ABB RAPID module: M_178.mod

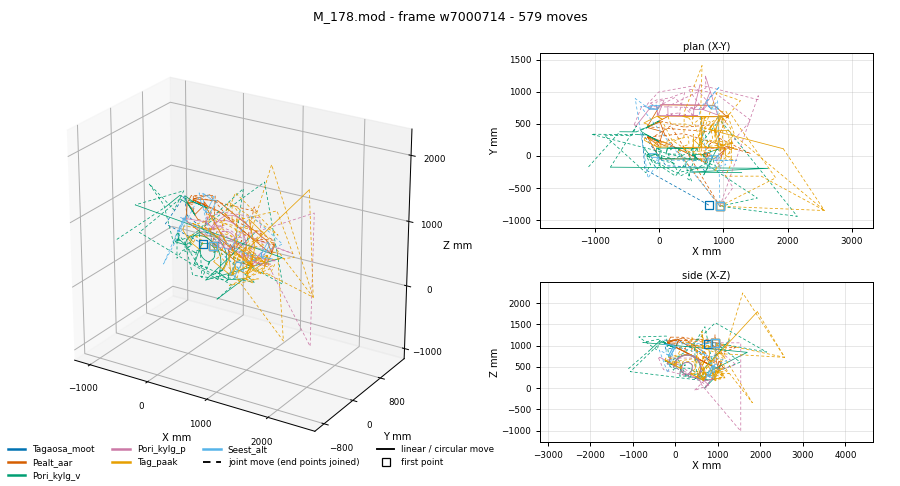
[picture p0: tool path of M_178.mod in frame w7000714, 579 of 583 moves have a stored position in this frame; points joined in program order, loops and branches not executed]
MODULE HITS_P

TASK PERS wobjdata w7000714:=[FALSE,FALSE,"STN2",[[0,0,0],[1,0,0,0]],[[375.036068751363,-383.154606661982,156.369033292662],[0.707106781186547,2.71584596430043E-17,2.9305070426361E-17,0.707106781186548]]];
CONST robtarget mooduli_vahetus := [[944.98,-783.48,1066.49],[0.140873,0.0138616,0.989908,-0.00676465],[0,-1,0,0],[358.608,-0.00699401,0.0391992,9E+09,9E+09,9E+09]];
CONST robtarget mooduli_vahetu10:=[[-90.91,322.81,1276.86],[0.262384,-0.0974996,0.959945,-0.0125037],[0,-1,0,0],[122.138,-6.09681,44.9368,9E+09,9E+09,9E+09]];
CONST robtarget mooduli_vahetu20:=[[3.88,808.65,1089.11],[0.234461,-0.125171,0.933949,-0.238956],[1,-1,0,0],[122.138,-6.09681,44.937,9E+09,9E+09,9E+09]];
TASK PERS pose VE1 := [[-6.83543,-0.0174255,-0.579834],[1,0,0,0]];
TASK PERS pose PE1 := [[0.5466,-0.00140381,0.050415],[1,0,0,0]];
TASK PERS pose VK1 := [[-0.057518,-0.763161,-0.332397],[1,0,0,0]];
TASK PERS pose VK2 := [[0.0793457,0.896591,0.228455],[1,0,0,0]];
TASK PERS pose VKs1 := [[1,2,0],[1,0,0,0]];
TASK PERS pose PEs1 := [[0,3,0],[1,0,0,0]];
TASK PERS pose PE2 := [[0,2,0],[1,0,0,0]];
TASK PERS pose VE2 := [[0,2,0],[1,0,0,0]];
TASK PERS pose VP1 := [[0.214996,0.419937,-0.887817],[1,0,0,0]];

  !**********************************************************
  !
  ! (c) Norcar-BSB Eesti AS
  !
  !**********************************************************
  !
  ! Moodul:       	7000714
  !
  ! Autor:   		Martins, Erki, Kert
  !
  ! Description:  	7000714 a60 tagaosa keevitusprogramm
  !
  ! Protseduurid:   	m??tmine enne keevitust smartac
  !
  ! Funktsioonid:    	m??tmine, keevitamine
  !
  ! Kuup?ev:      	04.03.2010
  !
  ! Versioon:      	0.7
  !
  ! Rakised:		a60 tagaosa rakis
  !
  ! Ajalugu:      	0.1 alustatud proge kirjutamist 04.03.2010
  !                 	0.2 esimene moodul tehtud 29.03.2010
  !				0.3 teine ja kolmas moodul tehtud 31.03.2010
  !				0.4 paagi mooduli tegemine 07.04.2010
  !				0.5 programmi korrastamine 08.04.2010
  !                	0.6 keevitusparameetrid sisse ja katsed 09.04.2010
  !				0.7 teise ringi katsetamine ja viies moodul
  !				0.8
  !
  !************************************************************

PROC HitsPMain()
	ActUnit STN2;
	Reset aDoRobHome;
	DRW_Number:="7000714";
	IF aDiK??ntP?ytOK=0 TPWrite "Waiting for turntables to reach home position";
	WaitDI aDiK??ntP?ytOK,1;

	TPErase;
	TPWrite "Traktori a60 tagaosa keevitus 7000714";
	TPWrite "versioon 0.7, 09.04.2010";

	! Parem pool valida tagant pool vaadates
	! rakise kaldenurk 27,3 kraadi

	! keevitusparameetrid: wld70v12sh24 ?huke plekk
	! weld100v10sh16 porilaud ja ??r kokku, l?hikesed ?mblused
	! wld100v5sh12 kere ja porilaud
	! wld200v10sh14 ots ja kere
	! wld250v6sh11 tugevdusribi
	! weld250v10sh11 korpus ja kaitseraud
	! wld200v6sh16 paksemad plaadid
	! wld200v8sh14 puksid, ring?mblused

start:
TPReadFK reg1,"Tee oma valik","M??da","Keevita","L?peta","","";

IF reg1=1 THEN
       GOTO yks;
ELSEIF reg1=2 THEN
       GOTO alusta;
ELSEIF reg1=3 THEN
       GOTO end;
    ENDIF

yks:
	Tagaosa_moot;
	GOTO start;

alusta:
Stop;

	! Moodul 1
	! Pealt perimeeter ja paagid kokku
	Pealt_aar;

	! Puhastus
	PuhdistRutWeld;

	! Moodul 2
	! Porilaud ja k?ljed vasakult
	!Stop;
	Pori_kylg_v;

	! Puhastus
	PuhdistRutWeld;

	! Moodul 3
	!Stop;
	! Porilaud ja k?ljed paremalt
	Pori_kylg_p;

	! Puhastus
	PuhdistRutWeld;

	! Moodul 4
	! tagaots ja paak seest
	Tag_paak;

	! Puhastus
	PuhdistRutWeld;

	! Moodul 5
	! V?ljast kinnitused ja alt puksid
	!Stop;
	Seest_alt;

	! Puhastus
	PuhdistRutWeld;

	GOTO end;
end:

MoveJ pHomeS2, v500, fine, tPKI500;
    DeactUnit STN2;
    RETURN;
ENDPROC


! M??tmine
PROC Tagaosa_moot()

	Stop;
	MoveJ [[771.19,-764.83,1049.41],[0.17262,-0.011269,0.984924,0.00151479],[0,-1,0,0],[358.606,0.00534949,0.0600025,9E+09,9E+09,9E+09]], v600, z200, tPKI500\WObj:=w7000714;

	! M??tmine smarttaciga ja pdisp kasutamine

	PDispOff;

	! Search - PROOV m??dab tagaosa

	!eest tagasapikkuse m66t
	MoveJ [[-222.07,-210.04,919.03],[0.387473,-0.533268,-0.439373,-0.610281],[1,-1,-2,0],[33.7138,0.00525396,0.0596227,9E+09,9E+09,9E+09]], v600, z200, tPKI500\WObj:=w7000714;
	Search_1D VE1, [[-281.87,349.61,976.70],[0.455775,-0.478529,-0.500064,-0.559657],[0,-1,-2,0],[33.7116,0.00531128,0.0594539,9E+09,9E+09,9E+09]], [[-245.65,349.67,979.75],[0.456433,-0.47783,-0.499358,-0.560349],[0,-1,-2,0],[33.7116,0.00531128,0.0592429,9E+09,9E+09,9E+09]], v600, tPKI500\WObj:=w7000714;
	Search_1D PE1, [[-279.88,515.34,977.24],[0.455844,-0.478471,-0.499981,-0.559725],[0,-1,-2,0],[33.7116,0.00531128,0.0593273,9E+09,9E+09,9E+09]], [[-250.66,515.16,979.95],[0.456426,-0.477841,-0.499362,-0.560342],[0,-1,-2,0],[33.7112,0.00525396,0.0593273,9E+09,9E+09,9E+09]], v600, tPKI500\WObj:=w7000714;
	MoveJ [[-271.44,361.19,1131.71],[0.456425,-0.477848,-0.499367,-0.560332],[0,-1,-2,0],[33.7116,0.00531128,0.0594539,9E+09,9E+09,9E+09]], v600, z200, tPKI500\WObj:=w7000714;

	!Vasaku kulje m66tmine
	MoveJ [[105.72,-153.88,1105.54],[0.108349,-0.674265,0.730311,-0.0165769],[0,0,-1,0],[33.7125,0.00534949,0.0591586,9E+09,9E+09,9E+09]], v600, z200, tPKI500\WObj:=w7000714;
	Search_1D VK1, [[120.39,-78.73,857.25],[0.0242109,0.669444,-0.741611,-0.0356805],[0,0,-1,0],[33.7132,0.00531128,0.0591586,9E+09,9E+09,9E+09]], [[121.03,-69.16,861.51],[0.0222677,0.66942,-0.741686,-0.03584],[0,0,-1,0],[33.7129,0.00534949,0.0591586,9E+09,9E+09,9E+09]], v600, tPKI500\WObj:=w7000714;
	MoveJ [[657.53,-174.78,809.55],[0.0222674,0.669428,-0.741679,-0.0358406],[0,0,-1,0],[33.7119,0.00534949,0.0590742,9E+09,9E+09,9E+09]], v600, z200, tPKI500\WObj:=w7000714;
	Search_1D VK2, [[706.38,-87.21,543.09],[0.0241212,0.669347,-0.74167,-0.0363144],[0,0,-2,0],[33.7125,0.00534949,0.0591586,9E+09,9E+09,9E+09]], [[707.65,-71.68,547.01],[0.0222997,0.669456,-0.741652,-0.0358542],[0,0,-2,0],[33.7125,0.00534949,0.0591586,9E+09,9E+09,9E+09]], v600, tPKI500\WObj:=w7000714;
	MoveJ [[706.29,-234.46,900.27],[0.0223105,0.669463,-0.741645,-0.0358672],[0,0,-1,0],[33.7119,0.00531128,0.0591586,9E+09,9E+09,9E+09]], v600, z200, tPKI500\WObj:=w7000714;
	!
	!
	MoveJ [[706.29,-234.46,900.26],[0.0223165,0.669465,-0.741643,-0.0358642],[0,0,-1,0],[33.7129,0.00531128,0.0592429,9E+09,9E+09,9E+09]], v600, z200, tPKI500\WObj:=w7000714;
	!
	!
	!

ENDPROC


! Pealt perimeeter ja paagid kokku
PROC Pealt_aar()

MoveJ mooduli_vahetus, v600, z50, tPKI500\WObj:=w7000714;

! kallutab lauda 17 kraadi, telg 1
MoveJ [[180.24,469.35,1197.20],[0.0518904,-0.882291,0.437678,0.165258],[0,-2,1,0],[252.909,16.9763,0.0391992,9E+09,9E+09,9E+09]], v200, z50, tPKI500\WObj:=w7000714;

! Keevitus 1.5, pealt sisemine perimeeter, esimene ?mblus, 90 mm, vasakult, OK
MoveJ [[-106.16,285.70,1199.65],[0.365736,0.833576,-0.285271,-0.300015],[0,-2,1,0],[223.84,16.9756,0.0391992,9E+09,9E+09,9E+09]], v600, z50, tPKI500\WObj:=w7000714;
PDispSet VKs1;
ArcLStart [[-184.93,290.61,1062.16],[0.282147,0.91122,-0.00162775,-0.300115],[0,-2,1,0],[223.922,16.9756,0.0353171,9E+09,9E+09,9E+09]], v600, seam1, m178job63, fine, tPKI500\WObj:=w7000714;
ArcL [[-182.70,295.03,1059.96],[0.31567,0.897368,-0.0303764,-0.306858],[0,-1,1,0],[223.905,16.975,0.0354859,9E+09,9E+09,9E+09]], v600, seam1, m178job63, fine, tPKI500\WObj:=w7000714;
ArcL [[-181.16,297.14,1059.57],[0.343632,0.766621,-0.361756,-0.404157],[0,-1,1,0],[223.774,16.9772,0.0418576,9E+09,9E+09,9E+09]], v600, seam1, m178job63, fine, tPKI500\WObj:=w7000714;
ArcLEnd [[-107.54,258.50,1021.43],[0.343541,0.766447,-0.362409,-0.403981],[0,-1,1,0],[223.649,16.975,0.0421108,9E+09,9E+09,9E+09]], v600, seam1, m178job63, fine, tPKI500\WObj:=w7000714;
PDispOff;
!Stop;

! Keevitus 1.6, pealt sisemine perimeeter, teine ?mblus, 170 mm, vasakult, OK
MoveJ [[-21.88,220.27,1045.21],[0.344664,0.764827,-0.363237,-0.405348],[0,-1,1,0],[223.835,16.9754,0.0388194,9E+09,9E+09,9E+09]], v600, z50, tPKI500\WObj:=w7000714;
ArcLStart [[-37.58,223.17,985.34],[0.34387,0.766267,-0.362247,-0.404187],[0,-1,1,0],[223.715,16.9765,0.0378489,9E+09,9E+09,9E+09]], v600, seam1, m178job63, fine, tPKI500\WObj:=w7000714;
ArcLEnd [[83.74,158.59,921.84],[0.344,0.766329,-0.362082,-0.404106],[0,-1,1,0],[223.926,16.9761,0.0403807,9E+09,9E+09,9E+09]], v600, seam1, m178job63, fine, tPKI500\WObj:=w7000714;
MoveJ [[206.18,140.94,924.64],[0.344664,0.764847,-0.363211,-0.405332],[0,-1,1,0],[223.836,16.9754,0.038946,9E+09,9E+09,9E+09]], v600, z50, tPKI500\WObj:=w7000714;

! Keevitus 1.7, pealt sisemine perimeeter, kolmas ?mblus, 900 mm, vasakult, OK
MoveJ [[245.32,122.46,948.22],[0.428788,0.781292,-0.355324,-0.281904],[0,-2,1,0],[223.836,16.9754,0.0390304,9E+09,9E+09,9E+09]], v600, z50, tPKI500\WObj:=w7000714;
ArcLStart [[219.87,127.02,851.73],[0.430441,0.781418,-0.353698,-0.28108],[0,-2,1,0],[223.838,16.9791,0.036583,9E+09,9E+09,9E+09]], v600, seam1, m178job63, fine, tPKI500\WObj:=w7000714;
ArcL [[342.17,127.04,789.47],[0.429347,0.781714,-0.354074,-0.281457],[0,-2,1,0],[223.735,16.9768,0.0410137,9E+09,9E+09,9E+09]], v600, seam1, m178job63, fine, tPKI500\WObj:=w7000714;
ArcL [[409.75,126.28,753.72],[0.429439,0.781537,-0.354188,-0.281664],[0,-2,1,0],[223.879,16.9747,0.039579,9E+09,9E+09,9E+09]], v600, seam1, m178job63, fine, tPKI500\WObj:=w7000714;
ArcL [[602.52,125.87,654.64],[0.429815,0.781282,-0.354003,-0.28203],[0,-2,1,0],[223.76,16.9766,0.0403807,9E+09,9E+09,9E+09]], v600, seam1, m178job63, fine, tPKI500\WObj:=w7000714;
ArcL [[895.88,124.47,502.15],[0.430572,0.780641,-0.353814,-0.282886],[0,-2,1,0],[223.711,16.9752,0.0383975,9E+09,9E+09,9E+09]], v600, seam1, m178job63, fine, tPKI500\WObj:=w7000714;
ArcLEnd [[1023.79,124.57,438.15],[0.316212,0.827255,-0.461489,-0.0518623],[0,-2,1,0],[223.957,16.9767,0.0422796,9E+09,9E+09,9E+09]], v600, seam1, m178job63, fine, tPKI500\WObj:=w7000714;
!Stop;
MoveL [[964.69,-11.95,633.96],[0.365253,0.816264,-0.423133,-0.145816],[0,-2,1,0],[223.84,16.9754,0.0391148,9E+09,9E+09,9E+09]], v600, z50, tPKI500\WObj:=w7000714;
MoveJ [[935.24,302.49,1253.35],[0.268514,0.719805,-0.421181,-0.482067],[0,-2,1,0],[900.475,16.9763,0.038946,9E+09,9E+09,9E+09]], v600, z50, tPKI500\WObj:=w7000714;

! tagaosa liigutamine, p??ramine -180 ja kallutamine -17 kraadi
MoveJ [[933.23,364.67,1157.80],[0.156036,0.433261,-0.854217,-0.241355],[0,0,0,0],[900.473,0.0294633,-0.0224089,9E+09,9E+09,9E+09]], v200, z50, tPKI500\WObj:=w7000714;


! Keevitus 1.8, pealt sisemine perimeeter, 400+1000 mm, paremalt, OK
MoveJ [[-182.46,453.50,1113.53],[0.0239912,-0.818382,-0.566844,-0.0914538],[0,0,-1,0],[900.473,-17.0628,-180.01,9E+09,9E+09,9E+09]], v600, z50, tPKI500\WObj:=w7000714;
!PDispSet PEs1;
ArcLStart [[-181.60,450.94,1062.98],[0.503117,-0.413223,-0.733358,0.195723],[0,0,-2,0],[900.45,-17.0603,-180.002,9E+09,9E+09,9E+09]], v600, seam1, m178job63, fine, tPKI500\WObj:=w7000714;
ArcL [[145.59,620.57,892.53],[0.508981,-0.543619,-0.650043,0.151203],[0,-1,-1,0],[900.468,-17.0623,-180.011,9E+09,9E+09,9E+09]], v600, seam1, m178job63, fine, tPKI500\WObj:=w7000714;
!PDispOff;
ArcL [[189.40,619.81,872.09],[0.508359,-0.544165,-0.649758,0.152549],[0,-1,-1,0],[900.389,-17.0611,-180.01,9E+09,9E+09,9E+09]], v600, seam1, m178job63, fine, tPKI500\WObj:=w7000714;
ArcL [[963.08,613.27,470.38],[0.507653,-0.544392,-0.649926,0.153374],[1,-1,0,0],[900.441,-17.0625,-180.009,9E+09,9E+09,9E+09]], v600, seam1, m178job63, fine, tPKI500\WObj:=w7000714;
ArcLEnd [[1025.00,613.30,438.63],[0.324043,-0.564722,-0.758986,0.00524122],[1,-1,0,0],[900.51,-17.0616,-180.01,9E+09,9E+09,9E+09]], v600, seam1, m178job63, fine, tPKI500\WObj:=w7000714;
MoveL [[1079.67,612.90,617.47],[0.409142,-0.560838,-0.716391,0.0696263],[1,-1,0,0],[900.466,-17.0627,-180.01,9E+09,9E+09,9E+09]], v600, z50, tPKI500\WObj:=w7000714;
MoveJ [[819.08,483.11,649.57],[0.380352,-0.742193,-0.550233,-0.0415458],[1,-1,0,0],[900.473,-17.0628,-180.01,9E+09,9E+09,9E+09]], v600, z50, tPKI500\WObj:=w7000714;
!Stop;

! Keevitus 1.9, pealt v?limine perimeeter, 400+960+260 mm, paremalt, OK
MoveJ [[384.40,449.47,940.53],[0.521441,-0.593526,-0.607333,0.0835091],[1,-1,-1,0],[900.473,-17.0628,-180.01,9E+09,9E+09,9E+09]], v600, z50, tPKI500\WObj:=w7000714;
MoveJ [[46.17,534.77,1158.25],[0.600818,-0.379123,-0.690069,0.138168],[0,0,-2,0],[900.473,-25.7634,-166.314,9E+09,9E+09,9E+09]], v600, z50, tPKI500\WObj:=w7000714;
!PDispSet PE2;
!Stop;
ArcLStart [[-184.51,460.44,1069.91],[0.496644,-0.128395,-0.848,0.133251],[0,0,-2,0],[900.771,-25.7553,-166.306,9E+09,9E+09,9E+09]], v600, seam1, m178job64, fine, tPKI500\WObj:=w7000714;
ArcL [[-173.78,476.50,1064.44],[0.554302,-0.193481,-0.808682,0.0367356],[0,0,-2,0],[900.416,-25.7545,-166.312,9E+09,9E+09,9E+09]], v600, seam1, m178job64, fine, tPKI500\WObj:=w7000714;
ArcL [[7.04,779.24,972.40],[0.572647,-0.266003,-0.772129,0.071665],[0,0,-2,0],[900.468,-25.7619,-166.314,9E+09,9E+09,9E+09]], v600, seam1, m178job64, fine, tPKI500\WObj:=w7000714;
ArcL [[16.15,792.14,969.22],[0.546633,-0.32251,-0.771885,-0.0370876],[0,0,-2,0],[900.605,-25.7608,-166.312,9E+09,9E+09,9E+09]], v600, seam1, m178job64, fine, tPKI500\WObj:=w7000714;
ArcL [[17.29,792.63,968.97],[0.486097,-0.575984,-0.655473,-0.0480558],[0,0,-1,0],[900.465,-25.7615,-166.313,9E+09,9E+09,9E+09]], v600, seam1, m178job64, fine, tPKI500\WObj:=w7000714;
ArcL [[61.54,794.51,942.69],[0.486117,-0.575989,-0.655457,-0.0479974],[0,0,-1,0],[900.479,-25.7614,-166.313,9E+09,9E+09,9E+09]], v600, seam1, m178job64, fine, tPKI500\WObj:=w7000714;
!ArcL [[26.13,798.11,960.35],[0.484105,-0.561883,-0.669531,0.0407281],[0,0,-2,0],[900.564,-25.7615,-166.313,9E+09,9E+09,9E+09]], v600, seam1, m178job64, fine, tPKI500\WObj:=w7000714;
!PDispOff;
ArcL [[218.26,793.40,860.22],[0.440223,-0.59926,-0.666261,-0.0564766],[0,0,-1,0],[900.512,-22.7548,-167.365,9E+09,9E+09,9E+09]], v600, seam1, m178job64, fine, tPKI500\WObj:=w7000714;
ArcL [[462.67,790.42,734.13],[0.443653,-0.60729,-0.65239,-0.0935942],[0,0,-1,0],[900.43,-22.7561,-167.369,9E+09,9E+09,9E+09]], v600, seam1, m178job64, fine, tPKI500\WObj:=w7000714;
ArcL [[742.57,789.03,587.93],[0.462626,-0.587719,-0.662256,-0.0445244],[1,-1,-1,0],[900.527,-22.7574,-167.369,9E+09,9E+09,9E+09]], v600, seam1, m178job64, fine, tPKI500\WObj:=w7000714;
ArcL [[851.66,788.32,531.91],[0.452915,-0.692054,-0.556899,-0.0761225],[1,-1,0,0],[900.414,-22.756,-167.367,9E+09,9E+09,9E+09]], v600, seam1, m178job64, fine, tPKI500\WObj:=w7000714;
ArcL [[855.89,786.75,530.12],[0.309039,-0.756387,-0.542731,-0.194471],[1,-1,0,0],[900.592,-22.7566,-167.369,9E+09,9E+09,9E+09]], v600, seam1, m178job64, fine, tPKI500\WObj:=w7000714;
ArcL [[865.09,778.53,525.36],[0.240514,-0.776627,-0.559111,-0.162482],[1,-1,0,0],[900.34,-22.7565,-167.369,9E+09,9E+09,9E+09]], v600, seam1, m178job64, fine, tPKI500\WObj:=w7000714;
ArcL [[1023.44,637.84,443.03],[0.305172,-0.843887,-0.420352,-0.13428],[1,-1,0,0],[900.508,-21.6371,-168.17,9E+09,9E+09,9E+09]], v600, seam1, m178job64, fine, tPKI500\WObj:=w7000714;
ArcLEnd [[1028.26,628.31,439.23],[0.104333,-0.92647,-0.329608,-0.148755],[1,-1,1,0],[900.435,-21.637,-168.167,9E+09,9E+09,9E+09]], v600, seam1, m178job64, fine, tPKI500\WObj:=w7000714;
MoveL [[1077.12,631.65,580.85],[0.334968,-0.898779,-0.276011,-0.0617454],[1,-1,0,0],[900.462,-17.0628,-180.01,9E+09,9E+09,9E+09]], v600, z50, tPKI500\WObj:=w7000714;
!Stop;
MoveJ [[911.67,287.97,765.35],[0.263835,-0.727529,-0.625551,0.0988923],[1,-1,0,0],[900.476,-17.0627,-180.01,9E+09,9E+09,9E+09]], v600, z50, tPKI500\WObj:=w7000714;

!laua pooramine 0?;0? ja puhastus
MoveJ [[1416.30,39.74,954.05],[0.0989373,0.157025,-0.973447,0.134],[0,-1,0,0],[900.477,0.118753,0.0317303,9E+09,9E+09,9E+09]], v200, z50, tPKI500\WObj:=w7000714;
PuhdistRutWeld;

! laua p??ramine 0 ja 17 kraadi
MoveJ [[373.90,347.34,998.41],[0.117153,0.675178,-0.725187,0.0672047],[1,-1,0,0],[900.477,17.0189,0.0317303,9E+09,9E+09,9E+09]], v200, z50, tPKI500\WObj:=w7000714;

! Keevitus 1.16, pealt v?limine perimeeter, katkestusega, 400+960+260 mm, vasakult, OK
MoveJ [[-90.42,300.54,1139.12],[0.392371,0.593922,-0.666197,-0.222452],[1,-1,0,0],[900.477,17.0189,0.0318147,9E+09,9E+09,9E+09]], v600, z50, tPKI500\WObj:=w7000714;
MoveJ [[-7.26,155.27,1132.10],[0.55973,0.636495,-0.490279,-0.202987],[1,-1,1,0],[900.477,23.261,-19.6927,9E+09,9E+09,9E+09]], v600, z50, tPKI500\WObj:=w7000714;
!PDispSet VE2;
ArcLStart [[-180.99,293.89,1069.89],[0.361586,0.702678,-0.482614,-0.377604],[1,-2,1,0],[900.55,23.2609,-19.6886,9E+09,9E+09,9E+09]], v600, seam1, m178job64, fine, tPKI500\WObj:=w7000714;
ArcL [[-172.19,275.51,1065.82],[0.362528,0.703271,-0.480746,-0.377979],[1,-2,1,0],[900.472,23.2629,-19.6841,9E+09,9E+09,9E+09]], v600, seam1, m178job64, fine, tPKI500\WObj:=w7000714;
ArcL [[12.62,-41.24,969.35],[0.363305,0.702574,-0.478589,-0.381252],[1,-2,1,0],[900.464,23.2617,-19.681,9E+09,9E+09,9E+09]], v600, seam1, m178job64, fine, tPKI500\WObj:=w7000714;
ArcL [[13.93,-43.98,966.67],[0.490227,0.715866,-0.473325,-0.152242],[1,-1,1,0],[900.529,23.2631,-19.6823,9E+09,9E+09,9E+09]], v600, seam1, m178job64, fine, tPKI500\WObj:=w7000714;
ArcL [[17.76,-45.14,963.78],[0.490161,0.716042,-0.473108,-0.152305],[1,-1,1,0],[900.405,23.263,-19.6888,9E+09,9E+09,9E+09]], v600, seam1, m178job64, fine, tPKI500\WObj:=w7000714;
!PDispOff;
ArcL [[409.73,-46.28,760.58],[0.489184,0.715938,-0.472985,-0.15626],[1,-1,0,0],[900.468,23.2622,-19.688,9E+09,9E+09,9E+09]], v600, seam1, m178job64, fine, tPKI500\WObj:=w7000714;
ArcL [[452.01,-46.08,738.89],[0.489114,0.71587,-0.473171,-0.156229],[1,-1,0,0],[900.642,23.2626,-19.6822,9E+09,9E+09,9E+09]], v600, seam1, m178job64, fine, tPKI500\WObj:=w7000714;
ArcL [[837.00,-47.76,538.25],[0.479378,0.722246,-0.473393,-0.156391],[0,0,-1,0],[900.538,23.2626,-19.6881,9E+09,9E+09,9E+09]], v600, seam1, m178job64, fine, tPKI500\WObj:=w7000714;
ArcL [[851.61,-46.66,530.84],[0.423876,0.859284,-0.254656,-0.13081],[0,0,-1,0],[900.402,23.2616,-19.691,9E+09,9E+09,9E+09]], v600, seam1, m178job64, fine, tPKI500\WObj:=w7000714;
ArcL [[857.00,-42.95,528.28],[0.386827,0.86793,-0.301478,-0.0785747],[0,0,-1,0],[900.62,20.2871,-19.3544,9E+09,9E+09,9E+09]], v600, seam1, m178job64, fine, tPKI500\WObj:=w7000714;
ArcL [[1012.18,92.00,448.44],[0.339783,0.9362,-0.0832581,-0.0338601],[0,0,-1,0],[900.49,20.2809,-19.3547,9E+09,9E+09,9E+09]], v600, seam1, m178job64, fine, tPKI500\WObj:=w7000714;
ArcL [[1023.90,103.83,443.36],[0.30711,0.951266,0.025384,-0.0115288],[0,0,-1,0],[900.508,20.2817,-19.3543,9E+09,9E+09,9E+09]], v600, seam1, m178job64, fine, tPKI500\WObj:=w7000714;
ArcLEnd [[1028.97,114.26,441.04],[0.30716,0.951259,0.0250954,-0.011467],[0,0,-1,0],[900.484,20.2805,-19.3551,9E+09,9E+09,9E+09]], v600, seam1, m178job64, fine, tPKI500\WObj:=w7000714;
MoveJ [[1009.60,129.26,607.74],[0.344702,0.916928,-0.125824,-0.156824],[0,0,-1,0],[900.477,17.0188,0.0318147,9E+09,9E+09,9E+09]], v600, z50, tPKI500\WObj:=w7000714;
GOTO toruta;

! laua kallutamine 27,3 kraadi
MoveJ [[1162.57,122.71,472.36],[0.140864,0.966293,-0.206823,0.0605097],[0,0,-1,0],[900.479,27.2716,0.0316459,9E+09,9E+09,9E+09]], v200, z50, tPKI500\WObj:=w7000714;

! Keevitus 1.17, paagi ?litoru keevitus, D65, 205 mm, vasakult, OK
MoveJ [[761.07,123.30,678.14],[0.365414,0.711061,-0.597258,0.0644121],[1,-1,0,0],[900.479,27.2716,0.0317303,9E+09,9E+09,9E+09]], v600, z50, tPKI500\WObj:=w7000714;
MoveJ [[796.44,199.49,743.61],[0.0479302,0.973161,-0.128236,0.184981],[0,0,-2,0],[380.209,27.2717,0.0316459,9E+09,9E+09,9E+09]], v600, z50, tPKI500\WObj:=w7000714;
MoveJ [[687.10,23.33,635.41],[0.047942,0.973163,-0.128221,0.184975],[0,0,-2,0],[380.21,27.2717,0.0317303,9E+09,9E+09,9E+09]], v600, z50, tPKI500\WObj:=w7000714;
ArcLStart [[695.23,20.35,610.24],[0.0479757,0.973171,-0.128186,0.184952],[0,0,-2,0],[380.209,27.2718,0.0316459,9E+09,9E+09,9E+09]], v600, seam1, wld200v8sh14, fine, tPKI500\WObj:=w7000714;
ArcC [[703.68,41.46,605.91],[0.233173,0.884181,-0.372829,0.157648],[0,0,-1,0],[380.209,27.2718,0.0315615,9E+09,9E+09,9E+09]], [[724.22,51.48,595.17],[0.413668,0.677563,-0.590079,0.146955],[0,0,-1,0],[380.209,27.2717,0.0317303,9E+09,9E+09,9E+09]], v600, seam1, wld200v8sh14, fine, tPKI500\WObj:=w7000714;
ArcC [[744.31,37.77,584.31],[0.560827,0.279575,-0.774777,0.0838623],[0,-1,0,0],[380.211,27.2717,0.0318991,9E+09,9E+09,9E+09]], [[749.01,21.17,581.66],[0.605493,-0.100927,-0.789225,0.0178112],[0,-1,0,0],[380.211,27.2717,0.0319835,9E+09,9E+09,9E+09]], v600, seam1, wld200v8sh14, fine, tPKI500\WObj:=w7000714;
ArcC [[738.53,-3.73,586.77],[0.523729,-0.550732,-0.646299,-0.068564],[0,-1,1,0],[380.211,27.2717,0.0317303,9E+09,9E+09,9E+09]], [[720.80,-10.17,596.10],[0.382247,-0.798907,-0.44818,-0.121536],[0,-1,1,0],[380.209,27.2717,0.0318147,9E+09,9E+09,9E+09]], v600, seam1, wld200v8sh14, fine, tPKI500\WObj:=w7000714;
ArcCEnd [[702.53,-1.70,606.23],[0.217979,-0.937243,-0.220726,-0.159192],[0,0,2,0],[380.209,27.2717,0.0317303,9E+09,9E+09,9E+09]], [[694.97,21.51,610.10],[0.0305759,-0.983588,0.026777,-0.175798],[0,0,2,0],[380.209,27.2717,0.0318991,9E+09,9E+09,9E+09]], v600, seam1, wld200v8sh14, fine, tPKI500\WObj:=w7000714;
MoveJ [[677.39,22.28,657.51],[0.0305932,-0.983584,0.0267976,-0.175812],[0,0,2,0],[380.21,27.2717,0.0317303,9E+09,9E+09,9E+09]], v600, z50, tPKI500\WObj:=w7000714;
MoveJ [[715.23,21.87,731.36],[0.0314181,-0.983594,0.0257474,-0.175765],[0,0,2,0],[380.212,27.2718,0.0315615,9E+09,9E+09,9E+09]], v600, z50, tPKI500\WObj:=w7000714;

! keevitus 1.18 olitoru 2. keevitus. Sihtida korgemale.
ArcLStart [[748.47,20.52,697.24],[0.0284428,-0.989467,0.0292656,-0.138894],[0,0,2,0],[380.211,27.2719,0.0312661,9E+09,9E+09,9E+09]], v600, seam1, wld100v5sh12, fine, tPKI500\WObj:=w7000714;
ArcC [[753.90,3.52,693.53],[0.29512,-0.905936,-0.262022,-0.153394],[0,0,2,0],[380.212,27.2719,0.0314771,9E+09,9E+09,9E+09]], [[758.04,0.42,692.07],[0.378817,-0.848515,-0.341376,-0.141365],[0,0,1,0],[380.213,27.2719,0.0315615,9E+09,9E+09,9E+09]], v600, seam1, wld100v5sh12, fine, tPKI500\WObj:=w7000714;
ArcC [[780.52,-0.11,681.16],[0.555558,-0.48452,-0.674518,-0.0402726],[0,-1,1,0],[380.212,27.272,0.0314771,9E+09,9E+09,9E+09]], [[789.68,16.12,677.29],[0.605207,-0.15056,-0.780951,0.034251],[0,-1,0,0],[380.212,27.2721,0.0315615,9E+09,9E+09,9E+09]], v600, seam1, wld100v5sh12, fine, tPKI500\WObj:=w7000714;
ArcC [[782.12,40.39,684.13],[0.48532,0.491825,-0.717743,0.086131],[0,-1,0,0],[380.215,27.2721,0.0316459,9E+09,9E+09,9E+09]], [[766.85,42.10,690.36],[0.2943,0.775359,-0.532609,0.168922],[0,0,-1,0],[380.214,27.272,0.0316459,9E+09,9E+09,9E+09]], v600, seam1, wld100v5sh12, fine, tPKI500\WObj:=w7000714;
ArcCEnd [[752.38,30.72,696.63],[0.0823334,0.954908,-0.245845,0.144683],[0,0,-2,0],[380.213,27.272,0.0317303,9E+09,9E+09,9E+09]], [[749.81,18.20,698.25],[0.0187265,-0.982495,0.0795466,-0.167411],[0,0,-2,0],[380.209,27.2719,0.0316459,9E+09,9E+09,9E+09]], v600, seam1, wld100v5sh12, fine, tPKI500\WObj:=w7000714;
MoveJ [[725.98,-104.59,807.21],[0.0243497,-0.967141,0.0782152,-0.240685],[0,0,-2,0],[380.212,27.2719,0.0312661,9E+09,9E+09,9E+09]], v600, z50, tPKI500\WObj:=w7000714;

! manualis aeg 13:55, 100% kiirusel
toruta:
MoveL [[188.78,164.77,1182.32],[0.351757,0.903929,-0.102661,-0.220549],[1,0,-1,0],[900.477,24.9716,0.185371,9E+09,9E+09,9E+09]], v600, z50, tPKI500\WObj:=w7000714;
MoveL [[-169.35,308.67,1074.09],[0.0381361,0.973148,-0.0686915,-0.21636],[1,0,-1,0],[601.879,24.9739,0.1844,9E+09,9E+09,9E+09]], v600, z50, tPKI500\WObj:=w7000714;
!ArcLStart [[-183.69,306.62,1059.10],[0.216625,0.952263,-0.0566688,-0.207508],[1,0,-1,0],[601.881,24.9747,0.183134,9E+09,9E+09,9E+09]], v600, seam1, m178job65, fine, tPKI500\WObj:=w7000714;
!ArcLEnd [[2.47,207.72,962.29],[0.21669,0.952252,-0.0566252,-0.2075],[1,0,-1,0],[601.881,24.9755,0.18229,9E+09,9E+09,9E+09]], v600, seam1, m178job65, fine, tPKI500\WObj:=w7000714;
ArcLStart [[-182.87,310.51,1063.00],[0.119162,0.96529,-0.078063,-0.218912],[1,0,-1,0],[601.92,24.9753,0.18305,9E+09,9E+09,9E+09]], v600, seam1, m178job66, fine, tPKI500\WObj:=w7000714;
ArcLEnd [[6.15,210.21,963.61],[0.119106,0.965289,-0.0780147,-0.218965],[1,0,-1,0],[601.876,24.9747,0.183134,9E+09,9E+09,9E+09]], v600, seam1, m178job66, fine, tPKI500\WObj:=w7000714;
MoveL [[57.63,376.88,1060.42],[0.0744618,-0.973587,0.0548019,0.208764],[1,0,-2,0],[601.885,24.9742,0.184189,9E+09,9E+09,9E+09]], v600, z50, tPKI500\WObj:=w7000714;
!ArcLStart [[-183.72,439.06,1060.86],[0.0763297,-0.957028,0.0605975,0.273131],[1,0,-2,0],[601.907,24.976,0.184189,9E+09,9E+09,9E+09]], v600, seam1, m178job65, fine, tPKI500\WObj:=w7000714;
!ArcLEnd [[8.45,537.87,962.35],[0.07636,-0.957023,0.0606505,0.273127],[1,0,-2,0],[601.862,24.9747,0.185075,9E+09,9E+09,9E+09]], v600, seam1, m178job65, fine, tPKI500\WObj:=w7000714;
ArcLStart [[-182.22,441.27,1061.82],[0.0764125,-0.957017,0.0606314,0.273139],[1,0,-2,0],[601.961,24.9744,0.184527,9E+09,9E+09,9E+09]], v600, seam1, m178job66, fine, tPKI500\WObj:=w7000714;
ArcLEnd [[8.78,538.10,964.11],[0.076471,-0.957017,0.0606792,0.27311],[1,0,-2,0],[601.869,24.9748,0.183683,9E+09,9E+09,9E+09]], v600, seam1, m178job66, fine, tPKI500\WObj:=w7000714;
MoveL [[83.51,335.92,1126.36],[0.0768622,-0.956981,0.0607954,0.273103],[1,0,-2,0],[601.886,24.9746,0.183683,9E+09,9E+09,9E+09]], v600, z50, tPKI500\WObj:=w7000714;

MoveJ mooduli_vahetus, v600, z50, tPKI500\WObj:=w7000714;

ENDPROC


! Porilaud ja k?ljed vasakult
PROC Pori_kylg_v()

MoveJ mooduli_vahetus, v600, z50, tPKI500\WObj:=w7000714;

! laua p??ramine ja kallutamine, -90 ja -90 kraadi
MoveJ [[1527.56,-656.12,612.18],[0.566224,-0.414194,0.434686,0.564697],[0,-1,0,0],[358.609,-90.0158,-89.9705,9E+09,9E+09,9E+09]], v200, z50, tPKI500\WObj:=w7000714;

!alternatiivne porilaua keevitus.2.1
!Stop;
MoveJ [[572.96,-23.79,219.28],[0.459065,0.157412,-0.452009,-0.748445],[0,0,1,0],[358.617,-127.415,-89.6268,9E+09,9E+09,9E+09]], v200, z50, tPKI500\WObj:=w7000714;
ArcLStart [[534.08,14.60,253.95],[0.341392,0.170853,-0.504174,-0.774642],[0,0,1,0],[358.631,-127.415,-89.6265,9E+09,9E+09,9E+09]], v200, seam1, m178job67, fine, tPKI500\WObj:=w7000714;
ArcL [[556.25,-7.26,298.85],[0.341411,0.170778,-0.504216,-0.774623],[0,0,1,0],[358.607,-127.415,-89.6273,9E+09,9E+09,9E+09]], v200, seam1, m178job67, z50, tPKI500\WObj:=w7000714;
ArcL [[570.60,-22.33,326.15],[0.398708,0.10403,-0.486785,-0.770228],[0,0,1,0],[358.715,-125.025,-89.9773,9E+09,9E+09,9E+09]], v200, seam1, m178job67, z50, tPKI500\WObj:=w7000714;
ArcL [[590.63,-49.24,379.80],[0.300559,0.14792,-0.535628,-0.77517],[0,-1,1,0],[358.605,-125.008,-89.9726,9E+09,9E+09,9E+09]], v200, seam1, m178job67, z50, tPKI500\WObj:=w7000714;
ArcC [[597.94,-49.71,418.79],[0.286569,0.224149,-0.674233,-0.642687],[0,-1,1,0],[358.865,-104.881,-89.9757,9E+09,9E+09,9E+09]], [[598.61,-48.93,423.22],[0.284227,0.232138,-0.688042,-0.62604],[0,-1,1,0],[358.894,-102.63,-89.9763,9E+09,9E+09,9E+09]], v200, seam1, m178job67, z10, tPKI500\WObj:=w7000714;
ArcL [[602.32,-49.42,456.59],[0.314306,0.226082,-0.727143,-0.566889],[0,-1,1,0],[358.818,-90.0107,-89.974,9E+09,9E+09,9E+09]], v200, seam1, m178job67, z50, tPKI500\WObj:=w7000714;
ArcC [[583.65,-49.46,578.79],[0.160275,0.384548,-0.734707,-0.535389],[0,-1,1,0],[358.582,-90.0143,-89.9725,9E+09,9E+09,9E+09]], [[558.64,-47.82,631.38],[0.0916303,0.457456,-0.72589,-0.505395],[0,-1,1,0],[358.474,-90.0159,-89.9718,9E+09,9E+09,9E+09]], v200, seam1, m178job67, z10, tPKI500\WObj:=w7000714;
ArcC [[500.41,-48.22,704.55],[0.0154446,0.508368,-0.70911,-0.488352],[0,-1,1,0],[414.039,-90.0124,-89.9729,9E+09,9E+09,9E+09]], [[472.91,-49.06,728.10],[0.0130383,-0.528015,0.7,0.480657],[0,-1,1,0],[435.496,-90.0111,-89.9733,9E+09,9E+09,9E+09]], v200, seam1, m178job67, z10, tPKI500\WObj:=w7000714;
ArcL [[432.66,-46.01,752.17],[0.0667774,-0.558399,0.73443,0.379927],[0,-1,0,0],[443.011,-90.005,-89.9756,9E+09,9E+09,9E+09]], v200, seam1, m178job67, z50, tPKI500\WObj:=w7000714;
ArcC [[320.15,-46.42,786.93],[0.271762,-0.637158,0.678161,0.245507],[0,-1,0,0],[598.731,-90.0089,-89.9756,9E+09,9E+09,9E+09]], [[256.16,-45.59,788.22],[0.37078,-0.666657,0.626103,0.161513],[0,-1,0,0],[683.013,-90.011,-89.9755,9E+09,9E+09,9E+09]], v200, seam1, m178job67, z10, tPKI500\WObj:=w7000714;
ArcC [[183.61,-45.05,773.57],[0.459894,-0.686265,0.559954,0.0631717],[0,-1,0,0],[737.214,-90.0087,-89.9733,9E+09,9E+09,9E+09]], [[151.34,-43.43,760.98],[0.496966,-0.690827,0.524923,0.0154951],[0,-1,0,0],[762.548,-90.0076,-89.9722,9E+09,9E+09,9E+09]], v200, seam1, m178job67, z10, tPKI500\WObj:=w7000714;
ArcL [[104.73,-43.35,735.62],[0.496966,-0.690809,0.524948,0.0154404],[0,-1,0,0],[762.508,-90.0073,-89.9752,9E+09,9E+09,9E+09]], v200, seam1, m178job67, z50, tPKI500\WObj:=w7000714;
ArcC [[66.14,-43.24,707.43],[0.496896,-0.690774,0.525064,0.0153374],[0,-1,0,0],[762.523,-90.0076,-89.9751,9E+09,9E+09,9E+09]], [[29.74,-43.29,672.73],[0.496859,-0.690741,0.525143,0.0152965],[0,-1,0,0],[762.539,-90.0081,-89.975,9E+09,9E+09,9E+09]], v200, seam1, m178job67, z10, tPKI500\WObj:=w7000714;
ArcL [[26.42,-42.31,669.24],[0.575143,-0.706885,0.402383,-0.0872576],[0,-1,0,0],[762.391,-90.0085,-89.9797,9E+09,9E+09,9E+09]], v200, seam1, m178job67, z50, tPKI500\WObj:=w7000714;
ArcL [[-15.58,-9.41,605.64],[0.651434,-0.649324,0.372356,-0.123953],[0,-1,0,0],[762.375,-90.004,-89.9733,9E+09,9E+09,9E+09]], v200, seam1, m178job67, z50, tPKI500\WObj:=w7000714;
ArcLEnd [[-44.01,20.11,549.48],[0.627735,-0.674263,0.358668,-0.150587],[0,-1,0,0],[762.392,-90.0026,-89.9697,9E+09,9E+09,9E+09]], v200, seam1, m178job67, fine, tPKI500\WObj:=w7000714;
MoveJ [[-43.22,8.74,449.30],[0.663991,-0.6342,0.351128,-0.183348],[0,-1,0,0],[776.94,-90.0134,-89.9686,9E+09,9E+09,9E+09]], v200, z50, tPKI500\WObj:=w7000714;

MoveJ [[242.40,-118.53,544.35],[0.758664,-0.445906,0.0707378,-0.469674],[1,0,-1,0],[1427.62,-100.045,-85.4322,9E+09,9E+09,9E+09]], v600, fine, tPKI500\WObj:=w7000714;

! Keevitus 2.3, porilaud seest, 1210 mm, vasakult, OK
MoveJ [[37.81,-70.37,544.52],[0.716966,-0.0163454,-0.364518,-0.593987],[0,0,-2,0],[1009,-90.0122,-89.97,9E+09,9E+09,9E+09]], v600, fine, tPKI500\WObj:=w7000714;
MoveJ [[29.04,84.36,539.17],[0.507124,0.0969799,-0.48977,-0.70253],[0,0,-2,0],[1085.24,-90.0121,-89.97,9E+09,9E+09,9E+09]], v600, fine, tPKI500\WObj:=w7000714;
!Stop;
ArcLStart [[-29.88,122.94,542.89],[0.504484,0.0907541,-0.494967,-0.701618],[0,0,-2,0],[1085.24,-90.0122,-89.9713,9E+09,9E+09,9E+09]], v600, seam1, m178job68, fine, tPKI500\WObj:=w7000714;
ArcL [[10.00,122.87,621.62],[0.483251,0.0799276,-0.492671,-0.719275],[0,0,-2,0],[1085.24,-90.0122,-89.971,9E+09,9E+09,9E+09]], v600, seam1, m178job68, fine, tPKI500\WObj:=w7000714;
ArcC [[58.75,122.93,685.64],[0.485228,0.0583463,-0.513626,-0.705223],[0,0,-2,0],[1046.34,-90.0099,-89.9742,9E+09,9E+09,9E+09]], [[119.77,122.89,733.03],[0.491958,0.0421263,-0.533135,-0.687002],[0,0,-2,0],[1009,-90.0077,-89.9771,9E+09,9E+09,9E+09]], v600, seam1, m178job68, fine, tPKI500\WObj:=w7000714;
ArcC [[180.45,123.46,760.70],[0.564952,-0.058518,-0.45451,-0.686169],[0,0,-2,0],[1009,-90.0078,-89.9767,9E+09,9E+09,9E+09]], [[248.98,123.84,773.44],[0.628969,-0.163144,-0.360116,-0.669403],[0,0,-2,0],[1009,-90.0079,-89.9763,9E+09,9E+09,9E+09]], v600, seam1, m178job68, fine, tPKI500\WObj:=w7000714;
ArcC [[288.93,122.02,772.85],[0.647366,-0.19692,-0.324973,-0.660706],[0,0,-2,0],[1009,-90.0078,-89.9753,9E+09,9E+09,9E+09]], [[407.44,119.21,745.66],[0.691447,-0.299742,-0.217746,-0.620197],[0,0,-2,0],[1009,-90.0075,-89.9721,9E+09,9E+09,9E+09]], v600, seam1, m178job68, fine, tPKI500\WObj:=w7000714;
ArcL [[430.64,118.55,732.15],[0.691541,-0.296732,-0.21608,-0.622119],[0,0,-2,0],[1009,-90.0089,-89.9643,9E+09,9E+09,9E+09]], v600, seam1, m178job68, fine, tPKI500\WObj:=w7000714;
ArcL [[449.20,117.99,721.39],[0.699511,-0.322333,-0.187062,-0.60975],[0,0,-2,0],[1009,-90.0066,-89.9709,9E+09,9E+09,9E+09]], v600, seam1, m178job68, fine, tPKI500\WObj:=w7000714;
ArcC [[523.13,117.92,653.04],[0.717041,-0.389593,-0.103125,-0.568715],[0,0,-2,0],[1008.99,-90.0068,-89.9729,9E+09,9E+09,9E+09]], [[564.33,117.24,586.33],[0.724479,-0.438735,-0.0377625,-0.530299],[0,0,-1,0],[1008.99,-90.0068,-89.9745,9E+09,9E+09,9E+09]], v600, seam1, m178job68, fine, tPKI500\WObj:=w7000714;
ArcC [[582.55,117.02,535.79],[0.717174,-0.48665,0.0381723,-0.49737],[0,0,-1,0],[1008.99,-90.0077,-89.9739,9E+09,9E+09,9E+09]], [[591.35,116.37,447.22],[0.688918,-0.560779,0.158604,-0.431005],[0,0,-1,0],[1009,-90.0093,-89.9725,9E+09,9E+09,9E+09]], v600, seam1, m178job68, fine, tPKI500\WObj:=w7000714;
ArcC [[590.62,117.25,433.10],[0.684383,-0.575368,0.18668,-0.407092],[0,0,-1,0],[1009,-90.0097,-89.9724,9E+09,9E+09,9E+09]], [[578.25,117.74,373.69],[0.651778,-0.626599,0.305234,-0.298987],[0,-1,-1,0],[1009,-90.0111,-89.9718,9E+09,9E+09,9E+09]], v600, seam1, m178job68, fine, tPKI500\WObj:=w7000714;
ArcL [[565.13,117.16,338.83],[0.655118,-0.636528,0.320964,-0.250272],[0,-1,0,0],[1009,-90.0074,-89.9742,9E+09,9E+09,9E+09]], v600, seam1, m178job68, fine, tPKI500\WObj:=w7000714;
ArcLEnd [[519.77,117.37,257.70],[0.657274,-0.634859,0.31662,-0.254358],[1,-1,0,0],[1009,-90.0102,-89.9701,9E+09,9E+09,9E+09]], v600, seam1, m178job68, fine, tPKI500\WObj:=w7000714;
MoveJ [[475.96,51.94,227.74],[0.681735,-0.611101,0.258296,-0.308346],[1,-1,0,0],[1009,-90.0112,-89.9698,9E+09,9E+09,9E+09]], v600, fine, tPKI500\WObj:=w7000714;
GOTO kylgedeta;

! Keevitus 2.4, porilaua alt, paagi ??r, esimene ?mblus, 110 mm, vasakult
MoveJ [[465.32,-50.67,240.40],[0.683886,-0.463526,0.123264,-0.549774],[1,0,-1,0],[1009,-90.0112,-89.9699,9E+09,9E+09,9E+09]], v600, fine, tPKI500\WObj:=w7000714;
MoveJ [[524.47,15.63,238.78],[0.631075,-0.418258,0.202155,-0.621241],[1,0,-1,0],[1009,-90.0112,-89.97,9E+09,9E+09,9E+09]], v600, fine, tPKI500\WObj:=w7000714;
Stop;
ArcLStart [[525.67,27.16,250.80],[0.594258,-0.581154,0.310601,-0.461135],[1,0,-1,0],[1009,-90.0113,-89.9715,9E+09,9E+09,9E+09]], v600, seam1, weld100v20sh16, fine, tPKI500\WObj:=w7000714;
ArcLEnd [[524.80,119.04,250.65],[0.627743,-0.579673,0.234095,-0.463809],[1,0,-1,0],[1009,-90.0114,-89.9707,9E+09,9E+09,9E+09]], v600, seam1, weld100v20sh16, fine, tPKI500\WObj:=w7000714;
MoveJ [[508.30,110.24,243.70],[0.702153,-0.469346,0.116887,-0.522528],[1,0,-1,0],[1009,-90.0112,-89.9699,9E+09,9E+09,9E+09]], v600, fine, tPKI500\WObj:=w7000714;
MoveJ [[453.00,45.61,237.11],[0.702147,-0.469339,0.116895,-0.522539],[1,0,-1,0],[1009,-90.0112,-89.97,9E+09,9E+09,9E+09]], v600, fine, tPKI500\WObj:=w7000714;
!liiga kuum, hakkab voolama, kiirust t?stetud

! Keevitus 2.5, porilaua alt, paagi ??r, teine ?mblus, 110 mm, vasakult
MoveJ [[213.41,-47.17,327.46],[0.60909,-0.0260551,-0.364759,-0.703763],[1,0,-2,0],[1009,-90.0112,-89.9701,9E+09,9E+09,9E+09]], v600, fine, tPKI500\WObj:=w7000714;
MoveJ [[-16.07,19.37,522.48],[0.771147,-0.083143,-0.261202,-0.574626],[0,0,-2,0],[1009,-90.0112,-89.97,9E+09,9E+09,9E+09]], v600, fine, tPKI500\WObj:=w7000714;
ArcLStart [[-41.12,31.01,543.59],[0.770932,-0.0834438,-0.26122,-0.574862],[0,0,-2,0],[1009,-90.0115,-89.9704,9E+09,9E+09,9E+09]], v600, seam1, weld100v20sh16, fine, tPKI500\WObj:=w7000714;
ArcLEnd [[-40.85,123.63,544.01],[0.770929,-0.0834511,-0.261224,-0.574863],[0,0,-2,0],[1009,-90.0112,-89.9695,9E+09,9E+09,9E+09]], v600, seam1, weld100v20sh16, fine, tPKI500\WObj:=w7000714;
MoveJ [[10.67,82.85,525.40],[0.77561,-0.243363,-0.238139,-0.531502],[0,0,-2,0],[1009,-90.0112,-89.9701,9E+09,9E+09,9E+09]], v600, fine, tPKI500\WObj:=w7000714;
MoveJ [[8.68,-158.74,524.78],[0.77561,-0.243359,-0.238141,-0.531503],[0,0,-2,0],[1009,-90.0112,-89.97,9E+09,9E+09,9E+09]], v600, fine, tPKI500\WObj:=w7000714;
!liiga kuum, hakkab voolama, kiirust t?stetud

! laua p??ramine, -100 ja -85,4 kraadi
MoveJ [[-39.12,-202.56,423.43],[0.771263,-0.181649,-0.184232,-0.581564],[0,0,-2,0],[1009,-100.05,-85.43,9E+09,9E+09,9E+09]], v200, fine, tPKI500\WObj:=w7000714;

!Vasaku pohja moot
!MoveJ [[-277.64,-345.23,389.22],[0.690812,-0.694774,-0.021359,0.199032],[0,0,-1,0],[1009,-100.049,-85.4311,9E+09,9E+09,9E+09]], v600, fine, tPKI500\WObj:=w7000714;
!Search_1D VP1, [[-126.43,171.18,560.08],[0.702202,-0.694447,0.1155,0.10638],[0,0,-1,0],[1009,-100.049,-85.4309,9E+09,9E+09,9E+09]], [[-128.80,166.49,570.00],[0.702401,-0.694352,0.113627,0.107698],[0,0,0,0],[1009,-100.049,-85.431,9E+09,9E+09,9E+09]], v200, tPKI500\WObj:=w7000714;
!MoveJ [[-277.64,-345.22,389.21],[0.69081,-0.694776,-0.0213578,0.199031],[0,0,-1,0],[1009,-100.049,-85.431,9E+09,9E+09,9E+09]], v600, fine, tPKI500\WObj:=w7000714;
!MoveJ [[-39.12,-202.56,423.43],[0.771261,-0.181652,-0.184234,-0.581566],[0,0,-2,0],[1009,-100.05,-85.4299,9E+09,9E+09,9E+09]], v600, fine, tPKI500\WObj:=w7000714;

! Keevitus 2.6, alumine ??r, esimene ?mblus, 140 mm, vasakult, OK
!MoveJ [[-71.64,-21.72,489.97],[0.757558,-0.376268,-0.0230221,-0.532915],[1,0,-1,0],[1427.62,-100.048,-85.4321,9E+09,9E+09,9E+09]], v600, fine, tPKI500\WObj:=w7000714;
!PDispSet VP1;
!ArcLStart [[-35.03,26.15,538.17],[0.66314,-0.228213,-0.238402,-0.671811],[1,0,-2,0],[1427.62,-100.043,-85.4329,9E+09,9E+09,9E+09]], v600, seam1, weld100v12sh16, fine, tPKI500\WObj:=w7000714;
!ArcLEnd [[-32.02,116.50,535.33],[0.663108,-0.228251,-0.238387,-0.671835],[1,0,-2,0],[1427.62,-100.043,-85.4329,9E+09,9E+09,9E+09]], v600, seam1, weld100v12sh16, fine, tPKI500\WObj:=w7000714;
!PDispOff;
!MoveJ [[-175.53,14.80,582.81],[0.759251,-0.445619,0.0717698,-0.468841],[1,0,-1,0],[1427.62,-100.048,-85.4322,9E+09,9E+09,9E+09]], v600, fine, tPKI500\WObj:=w7000714;

! laua p??ramine, -103 ja -64 kraadi
MoveJ [[-181.73,19.34,600.43],[0.755999,-0.445162,0.0747956,-0.474028],[0,0,-1,0],[1427.62,-102.958,-63.9271,9E+09,9E+09,9E+09]], v200, fine, tPKI500\WObj:=w7000714;

! Keevitus 2.7, alumine ??r, teine ?mblus, 110 mm, vasakult, OK
!MoveJ [[-165.49,26.34,600.87],[0.639332,-0.416884,0.217415,-0.608436],[0,0,-1,0],[1427.62,-102.957,-63.9269,9E+09,9E+09,9E+09]], v200, fine, tPKI500\WObj:=w7000714;
ArcLStart [[-162.46,29.68,608.98],[0.857786,-0.279596,-0.0391856,-0.429528],[1,0,-2,0],[1427.62,-102.957,-63.929,9E+09,9E+09,9E+09]], v600, seam1, weld100v12sh16, fine, tPKI500\WObj:=w7000714;
ArcLEnd [[-41.42,27.65,544.45],[0.857751,-0.280326,-0.0391144,-0.42913],[1,0,-2,0],[1427.62,-102.957,-63.9289,9E+09,9E+09,9E+09]], v600, seam1, weld100v12sh16, fine, tPKI500\WObj:=w7000714;
MoveL [[-192.42,-14.82,573.99],[0.755854,-0.445306,0.0748956,-0.474109],[0,0,-1,0],[1427.63,-102.957,-63.9302,9E+09,9E+09,9E+09]], v600, fine, tPKI500\WObj:=w7000714;
ArcLStart [[-167.87,33.13,613.03],[0.527932,-0.481364,0.239966,-0.657263],[0,0,-1,0],[1427.62,-102.957,-63.9263,9E+09,9E+09,9E+09]], v600, seam1, weld100v12sh16, fine, tPKI500\WObj:=w7000714;
ArcLEnd [[-227.49,112.88,645.27],[0.554642,-0.52011,0.193627,-0.619974],[0,0,-1,0],[1427.62,-102.958,-63.9276,9E+09,9E+09,9E+09]], v600, seam1, weld100v12sh16, fine, tPKI500\WObj:=w7000714;
MoveJ [[-244.74,103.31,638.02],[0.61884,-0.453919,0.204996,-0.607432],[0,0,-1,0],[1427.62,-102.958,-63.9271,9E+09,9E+09,9E+09]], v600, fine, tPKI500\WObj:=w7000714;
MoveJ [[-134.83,-137.72,608.86],[0.61882,-0.453913,0.204995,-0.607457],[1,0,-1,0],[2001.45,-102.958,-63.9271,9E+09,9E+09,9E+09]], v600, fine, tPKI500\WObj:=w7000714;
MoveJ [[-208.32,-261.20,1225.12],[0.618811,-0.453908,0.204998,-0.607469],[0,0,-1,0],[2001.45,-102.958,-63.927,9E+09,9E+09,9E+09]], v600, fine, tPKI500\WObj:=w7000714;

!GOTO ilmaotsteta;
!lauap88ramine koos robotiga
MoveJ [[-855.75,322.95,1204.81],[0.448921,-0.21845,0.687158,-0.527793],[0,0,0,0],[2001.45,-106.666,-0.0184423,9E+09,9E+09,9E+09]], v600, fine, tPKI500\WObj:=w7000714;

!keevitus 2.75 eesmised otsad. sisemine+v2limine kylg kokku vasakult
MoveJ [[-425.20,318.51,895.69],[0.18778,-0.271143,0.890141,-0.314437],[0,0,0,0],[2001.45,-106.666,-0.0185267,9E+09,9E+09,9E+09]], v600, fine, tPKI500\WObj:=w7000714;
!ArcLStart [[-288.08,304.64,868.17],[0.351163,-0.247489,0.848817,-0.308132],[1,-1,0,0],[2001.46,-106.666,-0.0183579,9E+09,9E+09,9E+09]], v600, seam1, wld100v16sh16, fine, tPKI500\WObj:=w7000714;
!ArcLEnd [[-216.24,304.91,1006.42],[0.351112,-0.247491,0.848814,-0.308197],[1,0,0,0],[2001.45,-106.666,-0.0182314,9E+09,9E+09,9E+09]], v600, seam1, wld100v16sh16, fine, tPKI500\WObj:=w7000714;
!MoveL [[-220.03,294.58,1021.61],[0.351191,-0.247519,0.848796,-0.308132],[0,0,0,0],[2001.45,-106.666,-0.0184423,9E+09,9E+09,9E+09]], v600, fine, tPKI500\WObj:=w7000714;
!ArcLStart [[-207.15,304.39,1022.94],[0.35115,-0.247485,0.848803,-0.308188],[1,0,0,0],[2001.45,-106.666,-0.0186955,9E+09,9E+09,9E+09]], v600, seam1, wld100v16sh16, fine, tPKI500\WObj:=w7000714;
!ArcLEnd [[-184.07,305.32,1066.70],[0.351133,-0.247498,0.848803,-0.308199],[0,0,0,0],[2001.46,-106.666,-0.0184423,9E+09,9E+09,9E+09]], v600, seam1, wld100v16sh16, fine, tPKI500\WObj:=w7000714;
!MoveJ [[-338.66,294.45,1017.35],[0.351187,-0.247515,0.848792,-0.308153],[0,0,0,0],[2001.45,-106.666,-0.0185267,9E+09,9E+09,9E+09]], v600, fine, tPKI500\WObj:=w7000714;
!MoveJ [[-348.94,294.02,892.13],[0.351174,-0.247508,0.848798,-0.308157],[1,-1,0,0],[2001.45,-106.666,-0.0184423,9E+09,9E+09,9E+09]], v600, fine, tPKI500\WObj:=w7000714;
!ArcLStart [[-289.29,311.06,867.64],[0.291958,-0.373572,0.799347,-0.369121],[1,0,0,0],[2001.46,-106.664,-0.018147,9E+09,9E+09,9E+09]], v600, seam1, wld70v3sh19\Weave:=weave14, fine, tPKI500\WObj:=w7000714;
!ArcLEnd [[-215.15,310.26,1004.62],[0.291993,-0.373603,0.799287,-0.369191],[0,0,0,0],[2001.46,-106.664,-0.0184423,9E+09,9E+09,9E+09]], v600, seam1, wld70v3sh19\Weave:=weave14, fine, tPKI500\WObj:=w7000714;
!MoveL [[-220.94,302.73,1011.45],[0.128899,-0.255811,0.843948,-0.45354],[0,0,0,0],[2001.45,-106.666,-0.0183579,9E+09,9E+09,9E+09]], v600, fine, tPKI500\WObj:=w7000714;
!ArcLStart [[-206.88,309.65,1021.19],[0.291972,-0.373623,0.799272,-0.36922],[0,0,0,0],[2001.45,-106.664,-0.0187799,9E+09,9E+09,9E+09]], v600, seam1, wld70v3sh19\Weave:=weave14, fine, tPKI500\WObj:=w7000714;
!ArcLEnd [[-185.13,310.02,1064.46],[0.291959,-0.373629,0.799271,-0.369227],[0,0,-1,0],[2001.45,-106.664,-0.018147,9E+09,9E+09,9E+09]], v600, seam1, wld70v3sh19\Weave:=weave14, fine, tPKI500\WObj:=w7000714;
!MoveJ [[-442.49,302.97,1063.20],[0.18766,-0.271093,0.890141,-0.314553],[0,0,0,0],[2001.45,-106.663,-0.0182314,9E+09,9E+09,9E+09]], v600, fine, tPKI500\WObj:=w7000714;

!keevitus 2.75 eesmised otsad. sisemine+v2limine kylg kokku paremalt
!MoveJ [[-651.26,465.70,639.87],[0.347461,-0.236838,0.864362,0.275789],[1,-1,1,0],[2001.45,-106.662,-0.0186955,9E+09,9E+09,9E+09]], v600, fine, tPKI500\WObj:=w7000714;
!MoveJ [[-420.90,460.23,713.69],[0.587599,-0.177803,0.789349,-0.00653432],[1,-1,1,0],[2001.45,-106.661,-0.0185267,9E+09,9E+09,9E+09]], v600, fine, tPKI500\WObj:=w7000714;
!ArcLStart [[-367.20,464.36,726.73],[0.587592,-0.177801,0.789355,-0.0065426],[1,-1,1,0],[2001.45,-106.661,-0.0185267,9E+09,9E+09,9E+09]], v600, seam1, wld100v16sh16, fine, tPKI500\WObj:=w7000714;
!ArcL [[-342.20,463.41,776.41],[0.754691,-0.177759,0.629727,-0.047837],[1,-1,1,0],[2001.45,-106.661,-0.0186111,9E+09,9E+09,9E+09]], v600, seam1, wld100v16sh16, fine, tPKI500\WObj:=w7000714;
!ArcL [[-341.70,464.84,776.55],[0.713054,0.0761429,0.675848,-0.170258],[1,-1,1,0],[2001.45,-106.661,-0.0187799,9E+09,9E+09,9E+09]], v600, seam1, wld100v16sh16, fine, tPKI500\WObj:=w7000714;
!ArcLEnd [[-328.29,464.53,802.54],[0.713044,0.0761724,0.675845,-0.170299],[1,-1,1,0],[2001.45,-106.661,-0.0186955,9E+09,9E+09,9E+09]], v600, seam1, wld100v16sh16, fine, tPKI500\WObj:=w7000714;
!MoveL [[-369.20,488.37,744.41],[0.713039,0.0761878,0.675845,-0.170313],[1,-1,0,0],[2001.46,-106.661,-0.0186955,9E+09,9E+09,9E+09]], v600, fine, tPKI500\WObj:=w7000714;
!ArcLStart [[-367.19,461.77,726.73],[0.586963,-0.00798072,0.806801,-0.0669671],[1,-1,1,0],[2001.45,-106.661,-0.0186111,9E+09,9E+09,9E+09]], v600, seam1, wld70v3sh19\Weave:=weave14, fine, tPKI500\WObj:=w7000714;
!ArcLEnd [[-342.22,460.57,776.42],[0.754684,-0.177768,0.629732,-0.0478465],[1,-1,1,0],[2001.46,-106.661,-0.0186111,9E+09,9E+09,9E+09]], v600, seam1, wld70v3sh19\Weave:=weave14, fine, tPKI500\WObj:=w7000714;
!MoveL [[-536.47,462.06,717.79],[0.754684,-0.177771,0.629731,-0.0478573],[1,-1,1,0],[2001.46,-106.661,-0.0187799,9E+09,9E+09,9E+09]], v600, fine, tPKI500\WObj:=w7000714;
!MoveJ [[-437.17,466.16,985.98],[0.460857,-0.124042,0.859589,0.182571],[1,-1,1,0],[2001.45,-106.661,-0.0184423,9E+09,9E+09,9E+09]], v600, fine, tPKI500\WObj:=w7000714;
!MoveJ [[-331.38,449.57,844.09],[0.2423,-0.077426,0.944182,0.209327],[1,0,1,0],[2001.45,-106.661,-0.0183579,9E+09,9E+09,9E+09]], v600, fine, tPKI500\WObj:=w7000714;
!ArcLStart [[-321.92,459.88,806.01],[0.242292,-0.0773586,0.944186,0.209344],[1,0,1,0],[2001.45,-106.661,-0.0186955,9E+09,9E+09,9E+09]], v600, seam1, wld100v16sh16, fine, tPKI500\WObj:=w7000714;
!ArcL [[-312.58,459.66,822.85],[0.419915,-0.118465,0.879778,0.188759],[1,-1,1,0],[2001.45,-106.661,-0.0184423,9E+09,9E+09,9E+09]], v600, seam1, wld100v16sh16, fine, tPKI500\WObj:=w7000714;
!ArcLEnd [[-184.68,460.35,1064.74],[0.419907,-0.118449,0.879778,0.188787],[1,-1,1,0],[2001.45,-106.661,-0.0186111,9E+09,9E+09,9E+09]], v600, seam1, wld100v16sh16, fine, tPKI500\WObj:=w7000714;
!MoveL [[-317.94,420.09,873.73],[0.419908,-0.118456,0.879777,0.188782],[1,-1,1,0],[2001.45,-106.661,-0.0186111,9E+09,9E+09,9E+09]], v600, fine, tPKI500\WObj:=w7000714;
!ArcLStart [[-319.01,457.27,805.77],[0.242296,-0.0773482,0.944182,0.209357],[1,0,1,0],[2001.45,-106.661,-0.0186111,9E+09,9E+09,9E+09]], v600, seam1, wld70v3sh19\Weave:=weave14, fine, tPKI500\WObj:=w7000714;
!ArcL [[-308.30,456.94,825.46],[0.41991,-0.118457,0.879778,0.188773],[1,-1,1,0],[2001.45,-106.661,-0.0182735,9E+09,9E+09,9E+09]], v600, seam1, wld70v3sh19\Weave:=weave14, fine, tPKI500\WObj:=w7000714;
!ArcLEnd [[-184.11,457.39,1063.35],[0.4199,-0.118431,0.879782,0.188794],[1,-1,1,0],[2001.45,-106.661,-0.0184423,9E+09,9E+09,9E+09]], v600, seam1, wld70v3sh19\Weave:=weave14, fine, tPKI500\WObj:=w7000714;
MoveJ [[-355.21,468.05,1155.56],[0.437448,-0.0586888,0.842633,0.308492],[0,-1,1,0],[2001.46,-106.662,-0.0179782,9E+09,9E+09,9E+09]], v600, fine, tPKI500\WObj:=w7000714;
MoveJ [[-759.38,-174.56,1075.02],[0.270239,-0.113003,0.78849,-0.540819],[0,0,0,0],[2001.46,-106.662,-0.0183579,9E+09,9E+09,9E+09]], v600, fine, tPKI500\WObj:=w7000714;
MoveL [[1694.64,-193.02,843.38],[0.46909,0.500099,-0.691347,0.227807],[0,0,0,0],[2001.46,-0.125633,-0.0185267,9E+09,9E+09,9E+09]], v200, fine, tPKI500\WObj:=w7000714;
MoveL [[473.47,-251.37,226.97],[0.681736,-0.611099,0.258294,-0.30835],[1,-1,-1,0],[1009,-90.0111,-89.9696,9E+09,9E+09,9E+09]], v600, fine, tPKI500\WObj:=w7000714;
MoveL [[1283.14,-260.33,1137.99],[0.681734,-0.611098,0.258299,-0.308353],[0,0,-1,0],[1009,-90.0112,-89.9698,9E+09,9E+09,9E+09]], v600, fine, tPKI500\WObj:=w7000714;
tagasi:
!
MoveJ [[1502.45,-3.30,1218.96],[0.00212533,-0.00251889,0.999989,-0.00330666],[-1,-2,1,0],[779.405,-0.00724241,0.0392836,9E+09,9E+09,9E+09]], v600, fine, tPKI500;
PuhdistRutWeld;
!
MoveJ [[-1100.71,-169.96,456.07],[0.443555,0.0143023,0.704398,-0.553967],[0,0,0,0],[2001.47,-133.225,0.0313927,9E+09,9E+09,9E+09]], v200, fine, tPKI500\WObj:=w7000714;
MoveJ [[-613.68,376.86,877.83],[0.00731551,0.431445,0.12439,0.893493],[0,-2,0,0],[2386.85,-133.225,0.0313927,9E+09,9E+09,9E+09]], v600, fine, tPKI500\WObj:=w7000714;
MoveL [[-360.55,374.52,1116.87],[0.00731834,0.431447,0.124386,0.893493],[0,-2,0,0],[2386.85,-133.225,0.0313927,9E+09,9E+09,9E+09]], v600, fine, tPKI500\WObj:=w7000714;
MoveJ [[-194.39,435.86,1029.38],[0.00749266,0.428504,0.124472,0.894895],[1,-2,0,0],[2386.86,-133.599,-0.00308251,9E+09,9E+09,9E+09]], v600, fine, tPKI500\WObj:=w7000714;
ArcLStart [[-192.77,448.65,1033.37],[0.102449,-0.376408,-0.236326,-0.889928],[1,-1,-1,0],[2386.86,-133.598,-0.00249175,9E+09,9E+09,9E+09]], v600, seam1, m178job69, fine, tPKI500\WObj:=w7000714;
ArcLEnd [[-1.47,545.04,936.64],[0.219268,-0.387838,-0.175013,-0.877995],[1,-1,-1,0],[2386.87,-133.598,-0.00282933,9E+09,9E+09,9E+09]], v600, seam1, m178job69, fine, tPKI500\WObj:=w7000714;
MoveL [[-191.94,443.33,1036.29],[0.102572,-0.376354,-0.236376,-0.889924],[1,-1,-1,0],[2386.86,-133.598,-0.00291372,9E+09,9E+09,9E+09]], v600, fine, tPKI500\WObj:=w7000714;
!ArcLStart [[-193.62,447.69,1033.79],[0.102459,-0.376397,-0.236345,-0.889927],[1,-1,-1,0],[2386.86,-133.598,-0.00308251,9E+09,9E+09,9E+09]], v600, seam1, wld100v4sh16\Weave:=weave4, fine, tPKI500\WObj:=w7000714;
!ArcLEnd [[-5.02,542.84,937.74],[0.219361,-0.387804,-0.174988,-0.877992],[1,-1,-1,0],[2386.87,-133.598,-0.00274493,9E+09,9E+09,9E+09]], v600, seam1, wld100v4sh16\Weave:=weave4, fine, tPKI500\WObj:=w7000714;
!MoveL [[-191.78,445.95,1036.17],[0.10256,-0.376346,-0.236385,-0.889926],[1,-1,-1,0],[2386.87,-133.598,-0.00291372,9E+09,9E+09,9E+09]], v600, fine, tPKI500\WObj:=w7000714;
MoveL [[-293.48,409.97,1111.36],[0.102563,-0.376332,-0.236323,-0.889948],[1,-1,-1,0],[2386.87,-133.598,-0.00291372,9E+09,9E+09,9E+09]], v600, fine, tPKI500\WObj:=w7000714;
MoveL [[-277.68,379.24,1094.19],[0.0624907,-0.413229,0.260657,-0.870285],[1,-1,0,0],[2386.87,-133.598,-0.00282933,9E+09,9E+09,9E+09]], v600, fine, tPKI500\WObj:=w7000714;
ArcLStart [[-190.70,325.62,1036.49],[0.113679,0.351349,-0.253123,0.894182],[1,-2,0,0],[2386.89,-133.599,-0.00109924,9E+09,9E+09,9E+09]], v600, seam1, m178job69, fine, tPKI500\WObj:=w7000714;
ArcLEnd [[-6.93,227.53,939.86],[0.144184,0.342325,-0.256283,0.892382],[1,-2,0,0],[2386.88,-133.598,-0.0032513,9E+09,9E+09,9E+09]], v600, seam1, m178job69, fine, tPKI500\WObj:=w7000714;
MoveL [[-190.89,327.36,1038.01],[0.113038,0.35152,-0.25274,0.894304],[1,-2,0,0],[2386.87,-133.598,-0.00350448,9E+09,9E+09,9E+09]], v600, fine, tPKI500\WObj:=w7000714;
!ArcLStart [[-194.26,324.38,1035.96],[0.0408954,-0.389838,0.319216,-0.862819],[1,-1,0,0],[2386.87,-133.598,-0.00291372,9E+09,9E+09,9E+09]], v600, seam1, wld100v4sh16\Weave:=weave4, fine, tPKI500\WObj:=w7000714;
!ArcLEnd [[-7.44,221.94,939.84],[0.11966,0.349792,-0.249833,0.894937],[1,-2,0,0],[2386.87,-133.598,-0.00274493,9E+09,9E+09,9E+09]], v600, seam1, wld100v4sh16\Weave:=weave4, fine, tPKI500\WObj:=w7000714;
!MoveL [[-214.90,333.82,1049.16],[0.0409451,-0.389842,0.319161,-0.862835],[1,-1,0,0],[2386.87,-133.598,-0.00291372,9E+09,9E+09,9E+09]], v600, z50, tPKI500\WObj:=w7000714;
MoveL [[-329.63,331.87,1084.50],[0.0409333,-0.389834,0.31918,-0.862832],[1,-2,0,0],[2386.87,-133.598,-0.00274493,9E+09,9E+09,9E+09]], v600, z50, tPKI500\WObj:=w7000714;
MoveJ [[-1056.36,338.19,389.25],[0.0409524,-0.389836,0.319199,-0.862824],[1,-2,1,0],[2386.87,-133.598,-0.00308251,9E+09,9E+09,9E+09]], v600, z50, tPKI500\WObj:=w7000714;
GOTO l6pp;

!ilmaotsteta:

! laua p??ramine koos roboti liikumisega, -115 ja -64 kraadi, v?ike liikumine
MoveJ [[589.10,-78.49,186.40],[0.254314,-0.0789472,-0.309474,-0.912863],[1,0,-1,0],[2229.32,-114.954,-63.9249,9E+09,9E+09,9E+09]], v500, fine, tPKI500\WObj:=w7000714;

! Keevitus 2.8, paagi alumine ??r, 160+260+20 mm, vasakult
MoveJ [[521.16,6.34,242.70],[0.254319,-0.0789652,-0.309501,-0.912851],[1,0,-2,0],[2229.32,-114.953,-63.9249,9E+09,9E+09,9E+09]], v500, fine, tPKI500\WObj:=w7000714;
ArcLStart [[531.75,21.90,248.20],[0.253665,-0.0792166,-0.309322,-0.913072],[1,0,-2,0],[2229.32,-114.969,-63.8418,9E+09,9E+09,9E+09]], v600, seam1, weld100v12sh16, fine, tPKI500\WObj:=w7000714;
ArcL [[586.21,21.39,221.29],[0.255289,-0.0888317,-0.320238,-0.907957],[1,0,-2,0],[2229.32,-114.953,-63.9248,9E+09,9E+09,9E+09]], v600, seam1, weld100v12sh16, fine, tPKI500\WObj:=w7000714;
ArcL [[670.16,20.85,177.84],[0.255284,-0.0888995,-0.320224,-0.907956],[1,0,-2,0],[2229.32,-114.953,-63.9249,9E+09,9E+09,9E+09]], v600, seam1, weld100v12sh16, fine, tPKI500\WObj:=w7000714;
ArcL [[681.94,23.80,178.61],[0.376654,0.0374323,-0.34328,-0.859588],[1,0,-1,0],[2229.32,-114.953,-63.9252,9E+09,9E+09,9E+09]], v600, seam1, weld100v12sh16, fine, tPKI500\WObj:=w7000714;
ArcL [[874.59,92.93,210.40],[0.255291,-0.0889261,-0.320221,-0.907953],[1,0,-2,0],[2229.32,-114.953,-63.9254,9E+09,9E+09,9E+09]], v600, seam1, weld100v12sh16, fine, tPKI500\WObj:=w7000714;
ArcLEnd [[907.55,103.16,215.25],[0.193217,-0.1506,-0.274649,-0.929815],[1,0,-2,0],[2229.32,-114.953,-63.9254,9E+09,9E+09,9E+09]], v600, seam1, weld100v12sh16, fine, tPKI500\WObj:=w7000714;
MoveL [[883.51,86.61,202.00],[0.193217,-0.150582,-0.274656,-0.929816],[1,0,-2,0],[2229.32,-114.953,-63.9256,9E+09,9E+09,9E+09]], v600, fine, tPKI500\WObj:=w7000714;
MoveL [[693.06,-294.62,2.49],[0.193223,-0.150582,-0.274658,-0.929814],[1,0,-1,0],[2229.32,-114.953,-63.9262,9E+09,9E+09,9E+09]], v600, fine, tPKI500\WObj:=w7000714;
!ArcLStart [[668.10,22.87,178.65],[0.255287,-0.0888425,-0.320232,-0.907958],[1,0,-2,0],[2229.32,-114.953,-63.9253,9E+09,9E+09,9E+09]], v600, seam1, wld70v6sh19\Weave:=weave4, fine, tPKI500\WObj:=w7000714;
!ArcC [[673.54,23.97,177.73],[0.23214,-0.14169,-0.338667,-0.900745],[1,0,-2,0],[2229.32,-114.953,-63.9247,9E+09,9E+09,9E+09]], [[682.11,25.64,179.13],[0.223607,-0.151384,-0.335653,-0.902453],[1,0,-2,0],[2229.32,-114.953,-63.9247,9E+09,9E+09,9E+09]], v600, seam1, wld70v6sh19\Weave:=weave4, fine, tPKI500\WObj:=w7000714;
!ArcL [[874.21,94.71,210.07],[0.224023,-0.141825,-0.325454,-0.907623],[1,0,-2,0],[2229.32,-114.953,-63.9247,9E+09,9E+09,9E+09]], v600, seam1, wld70v6sh19\Weave:=weave4, fine, tPKI500\WObj:=w7000714;
!ArcL [[902.77,101.62,213.25],[0.154022,-0.21411,-0.299997,-0.916754],[1,0,-2,0],[2229.32,-114.953,-63.9255,9E+09,9E+09,9E+09]], v600, seam1, wld70v6sh19\Weave:=weave4, fine, tPKI500\WObj:=w7000714;
!ArcLEnd [[916.39,109.12,217.58],[0.151434,-0.235361,-0.324539,-0.90352],[1,0,-2,0],[2229.33,-114.952,-63.9227,9E+09,9E+09,9E+09]], v600, seam1, wld70v6sh19\Weave:=weave4, fine, tPKI500\WObj:=w7000714;
!MoveL [[900.03,94.17,198.96],[0.152037,-0.232743,-0.32593,-0.903596],[1,0,-2,0],[2229.32,-114.953,-63.9248,9E+09,9E+09,9E+09]], v600, fine, tPKI500\WObj:=w7000714;
! l?pp muuta, liiga l?kkav, ??letab l?bi

! laua p??ramine koos robotiga, -90 ja -64 kraadi
MoveJ [[814.43,-76.78,158.69],[0.152036,-0.232779,-0.325924,-0.90359],[1,0,-1,0],[1918.89,-90.0021,-63.9247,9E+09,9E+09,9E+09]], v300, fine, tPKI500\WObj:=w7000714;
! laua p??ramine koos robotiga, -90 ja -90 kraadi
kylgedeta:
MoveJ [[327.90,-312.34,469.63],[0.556609,-0.749818,0.168534,-0.315526],[0,0,-1,0],[1323.92,-90.002,-90.0296,9E+09,9E+09,9E+09]], v300, fine, tPKI500\WObj:=w7000714;

! Keevitus 2.9, h?dromootori plaat, esimene ?mblus, 120 mm, vasakult
MoveJ [[115.01,69.66,469.54],[0.479481,-0.807917,0.33667,-0.0634191],[1,-1,0,0],[1323.92,-90.002,-90.0298,9E+09,9E+09,9E+09]], v600, fine, tPKI500\WObj:=w7000714;
ArcLStart [[126.35,122.31,473.42],[0.454954,-0.810189,0.369557,-0.00628068],[1,-1,0,0],[1323.92,-90.0012,-90.0302,9E+09,9E+09,9E+09]], v600, seam1, m178job69, fine, tPKI500\WObj:=w7000714;
ArcLEnd [[179.19,120.90,578.54],[0.446379,-0.779523,0.429129,0.0945526],[1,-1,0,0],[1323.92,-90.002,-90.0303,9E+09,9E+09,9E+09]], v600, seam1, m178job69, fine, tPKI500\WObj:=w7000714;
MoveJ [[185.70,106.71,581.53],[0.516194,-0.784125,0.340894,-0.0498445],[0,-1,0,0],[1323.92,-90.002,-90.0298,9E+09,9E+09,9E+09]], v600, fine, tPKI500\WObj:=w7000714;
!Stop;
! kiirust maha

! Keevitus 2.10, h?dromootori plaat, teine ?mblus, 270 mm, vasakult
MoveJ [[179.45,95.54,586.82],[0.432986,-0.774446,0.44672,0.114889],[1,-1,0,0],[1323.93,-90.0005,-90.0298,9E+09,9E+09,9E+09]], v600, fine, tPKI500\WObj:=w7000714;
ArcLStart [[185.87,119.36,586.63],[0.320001,-0.725379,0.516157,0.324051],[1,-1,1,0],[1323.92,-90.0006,-90.0299,9E+09,9E+09,9E+09]], v600, seam1, m178job69, fine, tPKI500\WObj:=w7000714;
ArcL [[266.49,119.25,605.06],[0.250545,-0.676776,0.552937,0.416489],[1,-1,1,0],[1323.92,-90,-90.0299,9E+09,9E+09,9E+09]], v600, seam1, m178job69, fine, tPKI500\WObj:=w7000714;
ArcC [[342.65,118.83,590.38],[0.0863772,-0.534624,0.600547,0.58827],[1,-1,1,0],[1323.92,-90.0005,-90.0312,9E+09,9E+09,9E+09]], [[403.24,117.35,528.45],[0.100531,0.326535,-0.595798,-0.726839],[1,-1,2,0],[1323.92,-90.001,-90.0326,9E+09,9E+09,9E+09]], v600, seam1, m178job69, fine, tPKI500\WObj:=w7000714;
!ArcC [[402.71,116.33,524.31],[0.169379,0.260574,-0.576906,-0.755376],[1,-1,2,0],[1323.92,-90.0011,-90.0305,9E+09,9E+09,9E+09]], [[402.98,117.43,523.41],[0.104661,0.318849,-0.594759,-0.73051],[1,-1,2,0],[1323.92,-90.001,-90.0315,9E+09,9E+09,9E+09]], v600, seam1, weld200v4sh14, fine, tPKI500\WObj:=w7000714;
ArcLEnd [[402.30,117.37,519.22],[0.100528,0.326515,-0.595792,-0.726853],[1,-1,2,0],[1323.92,-90.001,-90.0321,9E+09,9E+09,9E+09]], v600, seam1, m178job69, fine, tPKI500\WObj:=w7000714;
MoveJ [[406.31,82.54,507.83],[0.0699865,0.338358,-0.589433,-0.730196],[1,-1,2,0],[1323.92,-90.001,-90.0297,9E+09,9E+09,9E+09]], v600, fine, tPKI500\WObj:=w7000714;
!Stop;
MoveJ [[403.31,78.13,519.75],[0.119902,0.312163,-0.543468,-0.769949],[1,-1,-2,0],[1323.92,-90.001,-90.0295,9E+09,9E+09,9E+09]], v600, fine, tPKI500\WObj:=w7000714;

! Keevitus 2.11, h?dromootori plaat, kolmas ?mblus, 260 mm, vasakult
ArcLStart [[402.74,118.02,522.63],[0.119912,0.312147,-0.543472,-0.769951],[1,-1,-2,0],[1323.92,-90.0009,-90.0295,9E+09,9E+09,9E+09]], v600, seam1, m178job69, fine, tPKI500\WObj:=w7000714;
ArcL [[389.04,117.54,429.74],[0.156879,0.258687,-0.533515,-0.789831],[1,-1,-2,0],[1323.92,-90.0011,-90.0294,9E+09,9E+09,9E+09]], v600, seam1, m178job69, fine, tPKI500\WObj:=w7000714;
ArcC [[378.31,118.20,406.32],[0.177727,0.228357,-0.52626,-0.799573],[1,-1,-2,0],[1323.93,-90.001,-90.0303,9E+09,9E+09,9E+09]], [[363.80,117.84,386.35],[0.19837,0.19588,-0.519015,-0.808025],[1,-1,-2,0],[1323.93,-90.001,-90.0309,9E+09,9E+09,9E+09]], v600, seam1, m178job69, fine, tPKI500\WObj:=w7000714;
ArcLEnd [[298.10,120.49,325.67],[0.310561,0.0883594,-0.545964,-0.773091],[1,0,-2,0],[1323.92,-90.0011,-90.0319,9E+09,9E+09,9E+09]], v600, seam1, m178job69, fine, tPKI500\WObj:=w7000714;
MoveJ [[298.27,93.47,306.85],[0.304665,0.243835,-0.562422,-0.728976],[1,-1,-2,0],[1323.93,-90.0012,-90.0313,9E+09,9E+09,9E+09]], v600, fine, tPKI500\WObj:=w7000714;
!Stop;
MoveJ [[325.52,27.55,280.17],[0.47231,-0.197976,-0.397538,-0.761376],[1,0,-2,0],[1323.92,-90,-90.0299,9E+09,9E+09,9E+09]], v600, fine, tPKI500\WObj:=w7000714;

! Keevitus 2.12, h?dromootori plaat, neljas ?mblus, 230 mm, vasakult
MoveJ [[106.81,29.10,287.44],[0.585319,-0.458504,-0.197885,-0.638763],[1,0,-1,0],[1323.92,-90,-90.0299,9E+09,9E+09,9E+09]], v600, fine, tPKI500\WObj:=w7000714;
ArcLStart [[127.41,122.16,470.56],[0.626171,-0.604472,-0.00159351,-0.492465],[0,0,-1,0],[1323.92,-90,-90.0298,9E+09,9E+09,9E+09]], v600, seam1, m178job69, fine, tPKI500\WObj:=w7000714;
ArcL [[130.91,122.75,460.69],[0.790657,-0.476645,0.126496,-0.362865],[1,-1,-1,0],[1323.92,-90.0001,-90.0297,9E+09,9E+09,9E+09]], v600, seam1, m178job69, fine, tPKI500\WObj:=w7000714;
ArcL [[158.97,122.09,394.00],[0.807177,-0.475182,0.0937665,-0.337456],[1,-1,-1,0],[1323.92,-89.9991,-90.0291,9E+09,9E+09,9E+09]], v600, seam1, m178job69, fine, tPKI500\WObj:=w7000714;
ArcC [[184.33,121.94,363.05],[0.781759,-0.371832,-0.0978767,-0.490933],[1,0,-1,0],[1323.92,-89.9995,-90.0295,9E+09,9E+09,9E+09]], [[224.59,121.19,336.62],[0.677411,-0.190648,-0.32114,-0.63375],[1,0,-2,0],[1323.92,-90.0002,-90.0298,9E+09,9E+09,9E+09]], v600, seam1, m178job69, fine, tPKI500\WObj:=w7000714;
ArcCEnd [[254.89,121.65,327.44],[0.667896,-0.148565,-0.36536,-0.631155],[1,0,-2,0],[1323.92,-89.9991,-90.0298,9E+09,9E+09,9E+09]], [[298.62,119.50,327.40],[0.648296,-0.0965483,-0.431822,-0.619614],[1,0,-2,0],[1323.93,-89.9975,-90.0299,9E+09,9E+09,9E+09]], v600, seam1, m178job69, fine, tPKI500\WObj:=w7000714;
MoveL [[310.60,108.57,321.58],[0.594764,-0.0864429,-0.454867,-0.657176],[1,0,-2,0],[1323.92,-90,-90.0299,9E+09,9E+09,9E+09]], v600, fine, tPKI500\WObj:=w7000714;
MoveJ [[504.76,-393.09,328.55],[0.594761,-0.0864537,-0.454869,-0.657176],[1,0,-2,0],[1323.92,-90.0001,-90.0301,9E+09,9E+09,9E+09]], v600, fine, tPKI500\WObj:=w7000714;
GOTO kylgedeta2;

! roboti eemale liikumine ja laua p??ramine -87 ja -90 kraadi
MoveJ [[441.83,-355.57,1042.45],[0.531224,-0.755349,0.37774,-0.0675454],[0,0,0,0],[1323.92,-86.859,-89.5649,9E+09,9E+09,9E+09]], v300, fine, tPKI500\WObj:=w7000714;

! laua p??ramine -60 ja -115 kraadi
MoveJ [[698.20,395.77,1445.54],[0.29347,-0.921733,0.253507,-0.0042888],[0,0,0,0],[1281.9,-60.0034,-115.024,9E+09,9E+09,9E+09]], v200, fine, tPKI500\WObj:=w7000714;

! Keevitus 2.13, tagant paagi ?mblus, weavega, 170 mm, vasakult, OK
MoveJ [[855.26,-115.22,671.73],[0.293465,-0.921734,0.253509,-0.00430256],[1,-1,0,0],[1281.9,-60.0026,-115.024,9E+09,9E+09,9E+09]], v600, fine, tPKI500\WObj:=w7000714;
MoveJ [[877.06,-159.93,372.27],[0.554507,-0.750216,-0.206853,-0.294808],[1,0,0,0],[1281.9,-60.0025,-115.024,9E+09,9E+09,9E+09]], v600, fine, tPKI500\WObj:=w7000714;
MoveJ [[752.26,-104.08,312.83],[0.825207,-0.456362,-0.193496,-0.270792],[1,-1,-1,0],[1281.9,-60.0025,-115.024,9E+09,9E+09,9E+09]], v600, fine, tPKI500\WObj:=w7000714;
ArcLStart [[733.77,-45.04,306.81],[0.825269,-0.456156,-0.193645,-0.270844],[1,-1,-1,0],[1281.9,-60.0027,-115.024,9E+09,9E+09,9E+09]], v600, seam1, wld50v3sh8\Weave:=weave4, fine, tPKI500\WObj:=w7000714;
ArcL [[707.28,-16.10,249.57],[0.916661,-0.300508,-0.0554124,-0.257602],[1,-1,-1,0],[1281.9,-60.0024,-115.024,9E+09,9E+09,9E+09]], v600, seam1, wld50v3sh8\Weave:=weave4, fine, tPKI500\WObj:=w7000714;
ArcLEnd [[676.43,22.44,178.32],[0.908791,-0.318278,-0.0712005,-0.260251],[1,-1,-1,0],[1281.9,-60.0025,-115.024,9E+09,9E+09,9E+09]], v600, seam1, wld50v3sh8\Weave:=weave4, fine, tPKI500\WObj:=w7000714;
MoveJ [[701.55,-45.80,189.74],[0.825228,-0.456289,-0.193557,-0.270805],[1,-1,-1,0],[1281.9,-60.0025,-115.024,9E+09,9E+09,9E+09]], v600, fine, tPKI500\WObj:=w7000714;
MoveJ [[753.44,-159.00,259.60],[0.825228,-0.456289,-0.193552,-0.27081],[1,-1,-1,0],[1281.9,-60.0025,-115.024,9E+09,9E+09,9E+09]], v600, fine, tPKI500\WObj:=w7000714;

! laua p??ramine -60 ja -70 kraadi
MoveJ [[266.89,-264.39,259.40],[0.658626,-0.495522,-0.00399679,-0.566264],[1,-1,-1,0],[1281.9,-60.0179,-69.9828,9E+09,9E+09,9E+09]], v200, fine, tPKI500\WObj:=w7000714;

! Keevitus 2.14, eest k?lje ?mblus, weavega, 170 mm, vasakult, OK
MoveJ [[71.20,-158.72,673.90],[0.710536,-0.600462,0.0533776,-0.362955],[1,-1,-1,0],[1281.9,-60.0177,-69.983,9E+09,9E+09,9E+09]], v600, fine, tPKI500\WObj:=w7000714;
MoveJ [[-117.89,-56.84,740.00],[0.715179,-0.642089,0.0335708,-0.27407],[1,-1,-1,0],[1281.9,-60.0177,-69.9831,9E+09,9E+09,9E+09]], v600, fine, tPKI500\WObj:=w7000714;
ArcLStart [[-108.10,-39.70,737.36],[0.715128,-0.641933,0.0333826,-0.274591],[1,-1,-1,0],[1281.9,-60.017,-69.9833,9E+09,9E+09,9E+09]], v600, seam1, wld50v3sh8\Weave:=weave4, fine, tPKI500\WObj:=w7000714;
ArcLEnd [[-156.85,28.04,606.37],[0.715168,-0.641854,0.0333382,-0.274679],[1,-1,-1,0],[1281.9,-60.0178,-69.9831,9E+09,9E+09,9E+09]], v600, seam1, wld50v3sh8\Weave:=weave4, fine, tPKI500\WObj:=w7000714;
MoveJ [[-157.73,-42.47,596.32],[0.715168,-0.642031,0.0335258,-0.274241],[1,-1,-1,0],[1281.9,-60.0177,-69.983,9E+09,9E+09,9E+09]], v600, fine, tPKI500\WObj:=w7000714;
MoveJ [[252.46,-313.80,863.55],[0.721086,-0.658767,0.0260638,-0.213032],[1,-1,-1,0],[1281.9,-60.0168,-69.9834,9E+09,9E+09,9E+09]], v600, fine, tPKI500\WObj:=w7000714;
!
! laua p??ramine koos robotiga, -33 ja -38 kraadi
MoveJ [[942.27,566.80,1538.22],[0.43025,-0.58229,0.609664,-0.322697],[0,-1,-1,0],[1281.9,-33.6792,-38.8586,9E+09,9E+09,9E+09]], v200, fine, tPKI500\WObj:=w7000714;
kylgedeta2:

! laua p??ramine, koos robotiga, -33 ja -38 kraadi
GOTO tagasi;
l6pp:
MoveJ [[2148.86,-940.42,849.25],[0.155075,0.0314474,-0.934431,0.319066],[0,-1,-1,0],[1281.9,0.00122225,0.0430392,9E+09,9E+09,9E+09]], v200, fine, tPKI500\WObj:=w7000714;

! aeg manualis 9:55, 100 % juures

MoveJ mooduli_vahetus, v600, z50, tPKI500\WObj:=w7000714;

ENDPROC


! Porilaud ja k?ljed paremalt
PROC Pori_kylg_p()

MoveJ mooduli_vahetus, v600, z50, tPKI500\WObj:=w7000714;

! laua p??ramine 90 ja -90 kraadi ja 125 ja -90 kraadi
MoveJ [[1541.02,938.19,1066.50],[0.104351,-0.690581,0.70937,0.0948936],[0,-1,0,0],[358.607,-0.00781564,-90.0272,9E+09,9E+09,9E+09]], v200, z50, tPKI500\WObj:=w7000714;
MoveJ [[1540.63,875.38,-1010.61],[0.570491,0.410636,-0.412812,0.579229],[0,-1,0,0],[358.608,124.97,-89.7478,9E+09,9E+09,9E+09]], v200, z50, tPKI500\WObj:=w7000714;

!alternatiiv keevitus 3.1 porilaua kaar yhe jutiga.
!Stop;
MoveJ [[633.31,1107.30,63.48],[0.318627,-0.364546,-0.427003,0.76371],[1,-1,-2,0],[936.947,124.994,-89.2955,9E+09,9E+09,9E+09]], v600, z50, tPKI500\WObj:=w7000714;
ArcLStart [[544.24,736.02,253.25],[0.018259,-0.360912,-0.465547,0.807884],[1,0,-2,0],[937.012,124.994,-89.3036,9E+09,9E+09,9E+09]], v600, seam1, m178job67, fine, tPKI500\WObj:=w7000714;
ArcL [[558.73,749.65,280.71],[0.0420425,-0.326175,-0.477699,0.814645],[1,0,-2,0],[937.219,124.994,-89.2977,9E+09,9E+09,9E+09]], v200, seam1, m178job67, z50, tPKI500\WObj:=w7000714;
ArcL [[583.32,773.75,325.51],[0.0992641,-0.273367,-0.481165,0.826982],[1,0,-2,0],[937,124.994,-89.294,9E+09,9E+09,9E+09]], v200, seam1, m178job67, z50, tPKI500\WObj:=w7000714;
ArcL [[605.24,799.86,379.74],[0.0749869,-0.329676,-0.525586,0.780674],[1,0,-2,0],[937.058,118.133,-89.297,9E+09,9E+09,9E+09]], v200, seam1, m178job67, z50, tPKI500\WObj:=w7000714;
ArcL [[606.79,799.96,387.34],[0.249882,-0.263325,-0.685113,0.631538],[1,0,-2,0],[935.39,89.995,-90.0305,9E+09,9E+09,9E+09]], v200, seam1, m178job67, z50, tPKI500\WObj:=w7000714;
ArcC [[614.98,799.25,447.67],[0.18036,-0.32553,-0.706075,0.602462],[1,0,-2,0],[935.448,89.9953,-90.0292,9E+09,9E+09,9E+09]], [[605.75,796.21,539.13],[0.0721819,-0.411916,-0.724255,0.548243],[1,0,-2,0],[935.538,89.9959,-90.027,9E+09,9E+09,9E+09]], v200, seam1, m178job67, z10, tPKI500\WObj:=w7000714;
ArcC [[592.33,796.76,584.26],[0.014927,-0.477384,-0.728173,0.491576],[1,0,-2,0],[936.175,89.9958,-90.0276,9E+09,9E+09,9E+09]], [[567.69,795.33,634.26],[0.0547732,0.549012,0.725481,-0.411417],[1,0,-2,0],[936.969,89.9958,-90.0282,9E+09,9E+09,9E+09]], v200, seam1, m178job67, z10, tPKI500\WObj:=w7000714;
ArcC [[449.18,796.67,751.00],[0.180121,0.61231,0.704717,-0.309852],[1,0,-1,0],[936.9,89.9949,-90.0289,9E+09,9E+09,9E+09]], [[373.27,797.45,779.64],[0.239836,0.635567,0.687065,-0.257832],[1,0,-1,0],[936.864,89.9945,-90.0291,9E+09,9E+09,9E+09]], v200, seam1, m178job67, z10, tPKI500\WObj:=w7000714;
ArcL [[341.15,796.85,786.74],[0.239939,0.63563,0.686948,-0.257891],[1,0,-1,0],[937.084,89.994,-90.0299,9E+09,9E+09,9E+09]], v200, seam1, m178job67, z50, tPKI500\WObj:=w7000714;
ArcC [[242.34,799.59,787.15],[0.377278,0.684319,0.598871,-0.175282],[1,0,-1,0],[936.909,89.9947,-90.0282,9E+09,9E+09,9E+09]], [[196.37,799.57,776.50],[0.435094,0.70259,0.547143,-0.133029],[1,0,-1,0],[936.824,89.995,-90.0278,9E+09,9E+09,9E+09]], v200, seam1, m178job67, z10, tPKI500\WObj:=w7000714;
ArcC [[136.21,799.91,750.57],[0.550877,0.736263,0.391351,0.0360218],[1,-1,0,0],[937.011,89.9941,-90.0254,9E+09,9E+09,9E+09]], [[120.28,800.58,741.22],[0.577213,0.736949,0.341787,0.0831515],[1,-1,0,0],[937.062,89.9939,-90.0247,9E+09,9E+09,9E+09]], v200, seam1, m178job67, z10, tPKI500\WObj:=w7000714;
ArcC [[52.83,801.67,687.12],[0.549616,0.740663,0.386447,-0.00123518],[1,-1,-1,0],[929.311,89.9959,-90.0309,9E+09,9E+09,9E+09]], [[42.85,800.90,676.60],[0.544489,0.740574,0.393509,-0.0152894],[1,0,-1,0],[928.025,89.9962,-90.0319,9E+09,9E+09,9E+09]], v200, seam1, m178job67, z10, tPKI500\WObj:=w7000714;
ArcL [[35.84,798.15,669.23],[0.681973,0.594946,0.42511,0.0153433],[1,0,-1,0],[761.795,89.9959,-90.0645,9E+09,9E+09,9E+09]], v200, seam1, m178job67, z50, tPKI500\WObj:=w7000714;
ArcL [[10.36,778.49,632.67],[0.680064,0.590806,0.43367,0.0198073],[1,0,-1,0],[762.08,89.9954,-90.0671,9E+09,9E+09,9E+09]], v200, seam1, m178job67, z50, tPKI500\WObj:=w7000714;
ArcL [[-16.26,751.40,582.27],[0.680251,0.590559,0.433686,0.0204154],[1,0,-1,0],[761.836,89.9956,-90.0615,9E+09,9E+09,9E+09]], v200, seam1, m178job67, z50, tPKI500\WObj:=w7000714;
ArcLEnd [[-32.91,738.45,554.11],[0.680307,0.589973,0.434318,0.0219908],[1,0,-1,0],[761.963,89.9975,-90.0655,9E+09,9E+09,9E+09]], v200, seam1, m178job67, fine, tPKI500\WObj:=w7000714;
MoveJ [[-50.24,836.93,527.75],[0.80885,0.512755,0.147743,0.247018],[1,0,0,0],[761.991,89.9958,-90.066,9E+09,9E+09,9E+09]], v200, z50, tPKI500\WObj:=w7000714;

! Keevitus 3.3, porilaud seest, 1210 mm, paremalt, OK
MoveJ [[74.12,871.33,568.46],[0.448629,-0.165146,-0.535402,0.696279],[0,-1,1,0],[246.228,90.0008,-90.0293,9E+09,9E+09,9E+09]], v600, fine, tPKI500\WObj:=w7000714;
!Stop;
ArcLStart [[-17.65,633.88,549.19],[0.416233,-0.20537,-0.560219,0.686097],[0,-1,1,0],[246.232,90.0016,-90.0287,9E+09,9E+09,9E+09]], v600, seam1, m178job68, fine, tPKI500\WObj:=w7000714;
ArcL [[13.30,631.47,613.02],[0.416277,-0.205383,-0.560238,0.686051],[1,-1,1,0],[246.228,90.0016,-90.0299,9E+09,9E+09,9E+09]], v600, seam1, m178job68, fine, tPKI500\WObj:=w7000714;
ArcC [[118.53,630.45,724.62],[0.531557,-0.0451503,-0.453297,0.714095],[1,-1,1,0],[246.24,90.0017,-90.0294,9E+09,9E+09,9E+09]], [[251.44,630.17,769.33],[0.613119,0.103451,-0.335803,0.707545],[1,-1,1,0],[246.251,90.0019,-90.0291,9E+09,9E+09,9E+09]], v600, seam1, m178job68, fine, tPKI500\WObj:=w7000714;
ArcC [[321.98,628.52,769.96],[0.644921,0.178679,-0.270118,0.692235],[1,-1,1,0],[246.242,90.0019,-90.0292,9E+09,9E+09,9E+09]], [[419.89,627.76,742.82],[0.678111,0.282421,-0.168934,0.657166],[1,-1,1,0],[246.225,90.0019,-90.0292,9E+09,9E+09,9E+09]], v600, seam1, m178job68, fine, tPKI500\WObj:=w7000714;
ArcL [[427.93,628.13,740.39],[0.688298,0.329578,-0.119834,0.635032],[1,-1,0,0],[246.237,90.0018,-90.0304,9E+09,9E+09,9E+09]], v600, seam1, m178job68, fine, tPKI500\WObj:=w7000714;
ArcL [[442.98,627.95,732.49],[0.689264,0.335201,-0.113869,0.632132],[1,-1,0,0],[246.238,90.0014,-90.0309,9E+09,9E+09,9E+09]], v600, seam1, m178job68, fine, tPKI500\WObj:=w7000714;
ArcC [[527.47,628.42,659.05],[0.69763,0.425908,-0.0101992,0.576031],[1,-1,0,0],[246.255,90.0019,-90.0292,9E+09,9E+09,9E+09]], [[575.53,628.58,577.06],[0.693234,0.49607,0.0768996,0.517136],[1,-1,0,0],[246.267,90.0024,-90.0277,9E+09,9E+09,9E+09]], v600, seam1, m178job68, fine, tPKI500\WObj:=w7000714;
ArcC [[598.37,627.96,458.28],[0.664316,0.587026,0.208302,0.413155],[0,-1,0,0],[246.252,90.0022,-90.028,9E+09,9E+09,9E+09]], [[568.99,629.43,337.04],[0.609255,0.658035,0.335061,0.289022],[0,0,-1,0],[246.238,90.0019,-90.0281,9E+09,9E+09,9E+09]], v600, seam1, m178job68, fine, tPKI500\WObj:=w7000714;
ArcL [[533.81,628.24,271.88],[0.596688,0.668058,0.356591,0.26553],[0,0,-1,0],[246.23,90.0018,-90.0296,9E+09,9E+09,9E+09]], v600, seam1, m178job68, fine, tPKI500\WObj:=w7000714;
ArcLEnd [[524.67,627.81,258.48],[0.596688,0.668051,0.356625,0.265501],[0,0,-1,0],[246.222,90.0015,-90.0293,9E+09,9E+09,9E+09]], v600, seam1, m178job68, fine, tPKI500\WObj:=w7000714;
MoveJ [[469.15,725.60,263.56],[0.653115,0.634591,0.30227,0.281726],[0,0,-1,0],[303.299,90.0012,-90.0322,9E+09,9E+09,9E+09]], v600, fine, tPKI500\WObj:=w7000714;
GOTO kyljeta;

! Keevitus 3.4, porilaua alt, paagi ??r, esimene ?mblus, 110 mm, paremalt, OK
MoveL [[507.80,745.92,235.42],[0.573118,0.40638,0.475275,0.529628],[0,0,-1,0],[303.298,90.001,-90.0269,9E+09,9E+09,9E+09]], v600, fine, tPKI500\WObj:=w7000714;
ArcLStart [[537.95,720.68,252.62],[0.622501,0.345021,0.409572,0.570706],[0,0,0,0],[303.297,90.001,-90.0272,9E+09,9E+09,9E+09]], v600, seam1, weld100v12sh16, fine, tPKI500\WObj:=w7000714;
ArcLEnd [[534.96,627.93,251.68],[0.635971,0.325527,0.388668,0.581817],[0,0,0,0],[303.299,90.001,-90.0272,9E+09,9E+09,9E+09]], v600, seam1, weld100v12sh16, fine, tPKI500\WObj:=w7000714;
MoveJ [[526.10,625.34,249.36],[0.634551,0.356639,0.420564,0.541554],[0,0,0,0],[303.297,90.0009,-90.027,9E+09,9E+09,9E+09]], v600, fine, tPKI500\WObj:=w7000714;

! Keevitus 3.5, porilaua alt, paagi ??r, teine ?mblus, 110 mm, paremalt, OK
MoveJ [[241.21,908.76,338.25],[0.762956,0.017187,0.0266515,0.645673],[0,0,0,0],[585.985,90.0009,-90.027,9E+09,9E+09,9E+09]], v600, fine, tPKI500\WObj:=w7000714;
MoveJ [[-31.25,763.31,511.02],[0.767516,-0.0527972,-0.0147392,0.638683],[0,0,0,0],[585.984,90.001,-90.0271,9E+09,9E+09,9E+09]], v600, fine, tPKI500\WObj:=w7000714;
ArcLStart [[-31.04,725.95,551.01],[0.705795,-0.0215789,-0.267222,0.65573],[1,-1,1,0],[585.988,90.001,-90.0273,9E+09,9E+09,9E+09]], v600, seam1, weld100v12sh16, fine, tPKI500\WObj:=w7000714;
ArcLEnd [[-30.86,631.81,549.16],[0.671669,0.0374095,-0.305977,0.673677],[1,-1,1,0],[585.987,90.001,-90.0274,9E+09,9E+09,9E+09]], v600, seam1, weld100v12sh16, fine, tPKI500\WObj:=w7000714;
MoveJ [[-23.73,671.59,474.94],[0.671682,0.0374153,-0.305982,0.673661],[1,-1,1,0],[585.987,90.001,-90.0273,9E+09,9E+09,9E+09]], v600, fine, tPKI500\WObj:=w7000714;
MoveJ [[-29.22,750.19,464.85],[0.763168,0.134473,-0.168479,0.609187],[1,-1,1,0],[585.986,90.001,-90.027,9E+09,9E+09,9E+09]], v600, fine, tPKI500\WObj:=w7000714;

! laua liigutamine 125 ja -104 kraadi
MoveJ [[-29.27,750.18,464.90],[0.73034,0.600195,0.270215,0.182632],[1,-1,0,0],[585.986,125.362,-104.184,9E+09,9E+09,9E+09]], v200, fine, tPKI500\WObj:=w7000714;

! Keevitus 3.6, esimese paagi alumine serv, 140+360 mm, paremalt, OK
! laud liigub keevitusel kaasa
MoveJ [[-39.14,776.36,519.59],[0.857347,0.391483,0.297278,0.152724],[0,0,-1,0],[91.8236,125.362,-104.184,9E+09,9E+09,9E+09]], v600, fine, tPKI500\WObj:=w7000714;
ArcLStart [[-34.22,730.99,552.20],[0.963203,0.253251,0.0899912,0.00248961],[0,1,-2,0],[91.8291,125.362,-104.184,9E+09,9E+09,9E+09]], v600, seam1, weld100v6sh16, fine, tPKI500\WObj:=w7000714;
!ArcL [[-148.46,731.37,614.86],[0.866233,0.352322,0.316973,0.158237],[0,0,-1,0],[91.8217,125.362,-104.184,9E+09,9E+09,9E+09]], v600, seam1, weld100v6sh16, fine, tPKI500\WObj:=w7000714;
ArcLEnd [[-152.08,731.41,615.51],[0.963211,0.253208,0.0900303,0.00248599],[0,1,-2,0],[91.8298,125.362,-104.184,9E+09,9E+09,9E+09]], v600, seam1, weld100v12sh16, fine, tPKI500\WObj:=w7000714;
ArcLStart [[-158.32,728.25,619.52],[0.849869,0.371833,0.330359,0.174147],[1,0,-1,0],[91.8291,125.362,-104.184,9E+09,9E+09,9E+09]], v600, seam1, weld100v8sh16\Weave:=weave2, fine, tPKI500\WObj:=w7000714;
!ArcL [[-154.94,729.08,619.53],[0.849869,0.371845,0.330346,0.174147],[1,0,-1,0],[91.8281,125.362,-104.184,9E+09,9E+09,9E+09]], v600, seam1, weld100v6sh16, fine, tPKI500\WObj:=w7000714;
ArcL [[-237.89,624.45,661.46],[0.763113,0.363318,0.46621,0.26136],[1,0,-1,0],[91.8414,126.316,-117.609,9E+09,9E+09,9E+09]], v600, seam1, wld100v8sh16\Weave:=weave2, fine, tPKI500\WObj:=w7000714;
ArcLEnd [[-365.27,463.30,727.74],[0.765838,0.355538,0.468993,0.259099],[1,0,-1,0],[91.8317,126.49,-122.515,9E+09,9E+09,9E+09]], v600, seam1, wld100v8sh16\Weave:=weave2, fine, tPKI500\WObj:=w7000714;
MoveL [[-388.88,488.48,705.61],[0.804895,0.295649,0.455089,0.240066],[1,0,-1,0],[91.8223,126.49,-122.515,9E+09,9E+09,9E+09]], v600, fine, tPKI500\WObj:=w7000714;
MoveJ [[-273.37,770.80,435.84],[0.804885,0.295622,0.455118,0.240074],[0,0,-1,0],[91.8255,126.49,-122.515,9E+09,9E+09,9E+09]], v600, fine, tPKI500\WObj:=w7000714;

! Keevitus 3.7, tagumise paagi alumine serv, 160+260+20 mm, paremalt
MoveJ [[510.94,755.25,223.87],[0.0439785,0.205939,0.455068,-0.865199],[1,0,-2,0],[1652,126.709,-126.216,9E+09,9E+09,9E+09]], v600, fine, tPKI500\WObj:=w7000714;
ArcLStart [[537.69,725.92,250.40],[0.0362646,0.00954435,0.348335,-0.93662],[1,0,-2,0],[1652,126.709,-126.216,9E+09,9E+09,9E+09]], v600, seam1, wld70v6sh19\Weave:=weave3, fine, tPKI500\WObj:=w7000714;
ArcLEnd [[680.88,723.57,177.03],[0.00409431,0.0583284,0.356195,-0.932581],[1,0,-2,0],[1652.01,126.709,-126.216,9E+09,9E+09,9E+09]], v600, seam1, wld70v6sh19\Weave:=weave3, fine, tPKI500\WObj:=w7000714;
MoveJ [[450.60,1041.36,-54.20],[0.00462524,0.0583077,0.35614,-0.932601],[1,0,-2,0],[1652,126.709,-126.216,9E+09,9E+09,9E+09]], v600, fine, tPKI500\WObj:=w7000714;
!Stop;

!GOTO tagantoblsetap;
!ArcLStart [[681.31,723.09,175.84],[0.00408424,0.0583176,0.356208,-0.932577],[1,0,-2,0],[1652,126.709,-126.216,9E+09,9E+09,9E+09]], v600, seam1, wld70v6sh19\Weave:=weave4, fine, tPKI500\WObj:=w7000714;
!ArcL [[868.65,650.63,205.76],[0.196747,0.356249,0.396173,-0.823059],[1,0,-2,0],[1652.01,126.709,-126.216,9E+09,9E+09,9E+09]], v600, seam1, wld70v6sh19\Weave:=weave4, z5, tPKI500\WObj:=w7000714;
!ArcLEnd [[911.63,633.46,213.34],[0.185741,0.325089,0.429768,-0.821656],[1,0,-2,0],[1652,126.709,-126.216,9E+09,9E+09,9E+09]], v600, seam1, wld70v6sh19\Weave:=weave4, fine, tPKI500\WObj:=w7000714;
!MoveL [[908.83,647.63,201.18],[0.169406,0.319195,0.450528,-0.816359],[1,0,-2,0],[1652,126.709,-126.216,9E+09,9E+09,9E+09]], v600, fine, tPKI500\WObj:=w7000714;
!MoveJ [[846.69,813.17,164.05],[0.245785,0.317662,0.529723,-0.747045],[1,0,-2,0],[1652,126.709,-126.216,9E+09,9E+09,9E+09]], v600, fine, tPKI500\WObj:=w7000714;
! muuta keevituse l?pp, hakkab l?ikama, programmeerida eraldi

! laua p??ramine koos robotiga, 116 ja -108 kraadi
MoveJ [[789.78,993.10,71.99],[0.245807,0.317666,0.52972,-0.747037],[1,0,-2,0],[1652,116.142,-107.994,9E+09,9E+09,9E+09]], v600, fine, tPKI500\WObj:=w7000714;
MoveJ [[789.45,992.32,72.29],[0.694989,0.630977,0.148413,0.31118],[1,-1,0,0],[1652,116.142,-107.994,9E+09,9E+09,9E+09]], v600, fine, tPKI500\WObj:=w7000714;
ArcLStart [[680.44,723.34,175.33],[0.89142,0.284089,-0.118793,0.332496],[1,-1,1,0],[1652,116.142,-107.994,9E+09,9E+09,9E+09]], v600, seam1, wld70v6sh19\Weave:=weave4, fine, tPKI500\WObj:=w7000714;
ArcL [[860.73,656.11,203.11],[0.880704,0.323697,-0.120456,0.324149],[1,-1,1,0],[1652,116.142,-107.994,9E+09,9E+09,9E+09]], v600, seam1, wld70v6sh19\Weave:=weave4, fine, tPKI500\WObj:=w7000714;
ArcLEnd [[908.17,637.93,210.48],[0.829515,0.375053,-0.00134834,0.413811],[1,-1,1,0],[1652,116.142,-107.994,9E+09,9E+09,9E+09]], v600, seam1, wld70v6sh19\Weave:=weave4, fine, tPKI500\WObj:=w7000714;
MoveL [[879.25,736.67,271.25],[0.829514,0.375055,-0.00134684,0.413812],[1,-1,1,0],[1652,116.142,-107.994,9E+09,9E+09,9E+09]], v600, fine, tPKI500\WObj:=w7000714;
MoveL [[719.73,1240.99,13.17],[0.829515,0.375057,-0.00134109,0.413807],[1,-1,1,0],[1652,116.142,-107.994,9E+09,9E+09,9E+09]], v600, fine, tPKI500\WObj:=w7000714;
!tagantoblsetap:

! laua p??ramine koos robotiga, 90 ja -90 kraadi
MoveJ [[726.48,1059.02,79.11],[0.727515,0.377491,0.558359,-0.128294],[1,0,-1,0],[1158.51,89.994,-90.0248,9E+09,9E+09,9E+09]], v200, fine, tPKI500\WObj:=w7000714;
kyljeta:

! Keevitus 3.8, h?dromootori plaat, esimene ?mblus, 120 mm, paremalt
MoveJ [[133.33,770.01,451.66],[0.439625,0.604002,0.664321,0.0242721],[1,0,-1,0],[553.979,89.994,-90.0249,9E+09,9E+09,9E+09]], v600, fine, tPKI500\WObj:=w7000714;
ArcLStart [[136.56,628.55,473.59],[0.427038,0.697091,0.572988,-0.058211],[1,0,-1,0],[553.979,89.9942,-90.0251,9E+09,9E+09,9E+09]], v600, seam1, m178job69, fine, tPKI500\WObj:=w7000714;
ArcLEnd [[195.35,627.62,587.70],[0.378093,0.688078,0.593203,-0.178066],[1,0,-1,0],[553.982,89.9951,-90.023,9E+09,9E+09,9E+09]], v600, seam1, m178job69, fine, tPKI500\WObj:=w7000714;
MoveL [[195.08,656.98,583.06],[0.464758,0.706669,0.532358,-0.0348653],[1,0,-1,0],[553.979,89.994,-90.0248,9E+09,9E+09,9E+09]], v600, fine, tPKI500\WObj:=w7000714;
! kuumem ja t?itvam z=8, a=5,6, praegu 4 ja 5 vahel

! Keevitus 3.9, h?dromootori plaat, teine ?mblus, 270 mm, paremalt
MoveL [[195.11,657.00,583.08],[0.264868,0.711073,0.557305,-0.337095],[1,0,-2,0],[553.979,89.994,-90.0249,9E+09,9E+09,9E+09]], v600, fine, tPKI500\WObj:=w7000714;
ArcLStart [[196.55,629.59,587.00],[0.226306,0.727765,0.562233,-0.320997],[1,0,-2,0],[553.992,89.9945,-90.0246,9E+09,9E+09,9E+09]], v600, seam1, m178job69, fine, tPKI500\WObj:=w7000714;
!ArcC [[198.13,629.63,587.87],[0.27613,0.752908,0.538611,-0.258423],[1,0,-1,0],[553.987,89.9941,-90.0248,9E+09,9E+09,9E+09]], [[208.05,629.26,591.48],[0.244878,0.738012,0.554268,-0.296921],[1,0,-2,0],[553.98,89.9941,-90.0248,9E+09,9E+09,9E+09]], v600, seam1, weld200v4sh14, z5, tPKI500\WObj:=w7000714;
ArcL [[273.46,628.82,606.06],[0.13738,0.670456,0.590784,-0.427307],[1,0,-2,0],[553.98,89.9942,-90.0256,9E+09,9E+09,9E+09]], v600, seam1, m178job69, fine, tPKI500\WObj:=w7000714;
ArcC [[342.27,627.58,595.02],[0.0120826,0.570869,0.608391,-0.551203],[1,0,-2,0],[553.979,89.9942,-90.0254,9E+09,9E+09,9E+09]], [[410.60,628.68,534.60],[0.148176,-0.402769,-0.59088,0.683142],[1,0,-2,0],[553.973,89.9942,-90.0257,9E+09,9E+09,9E+09]], v600, seam1, m178job69, z5, tPKI500\WObj:=w7000714;
ArcCEnd [[409.87,628.20,527.63],[0.198316,-0.349918,-0.575517,0.712046],[1,0,-2,0],[553.973,89.9943,-90.0253,9E+09,9E+09,9E+09]], [[409.25,628.61,523.49],[0.223146,-0.311323,-0.567683,0.728712],[1,0,-2,0],[553.975,89.9943,-90.0249,9E+09,9E+09,9E+09]], v600, seam1, m178job69, fine, tPKI500\WObj:=w7000714;
MoveL [[408.36,646.10,524.92],[0.257032,-0.266668,-0.55359,0.745897],[1,0,-3,0],[553.979,89.994,-90.0251,9E+09,9E+09,9E+09]], v600, fine, tPKI500\WObj:=w7000714;

! Keevitus 3.10, h?dromootori plaat, kolmas ?mblus, 260 mm, paremalt
ArcLStart [[412.03,629.68,525.23],[0.327163,-0.154111,-0.488539,0.794069],[1,0,-3,0],[553.973,89.9946,-90.0252,9E+09,9E+09,9E+09]], v600, seam1, m178job69, fine, tPKI500\WObj:=w7000714;
ArcL [[398.47,628.23,440.37],[0.357796,-0.10256,-0.466954,0.802134],[1,0,-3,0],[553.985,89.9942,-90.0249,9E+09,9E+09,9E+09]], v600, seam1, m178job69, fine, tPKI500\WObj:=w7000714;
ArcC [[386.51,628.37,411.12],[0.43175,0.02433,-0.404041,0.806072],[1,-1,-3,0],[553.983,89.9942,-90.0248,9E+09,9E+09,9E+09]], [[365.26,627.88,384.92],[0.496933,0.148332,-0.328504,0.789393],[1,-1,-3,0],[553.98,89.9943,-90.0248,9E+09,9E+09,9E+09]], v600, seam1, m178job69, z5, tPKI500\WObj:=w7000714;
ArcLEnd [[309.72,630.17,332.22],[0.526314,0.225351,-0.278863,0.771004],[1,-1,-3,0],[553.979,89.9942,-90.0257,9E+09,9E+09,9E+09]], v600, seam1, m178job69, fine, tPKI500\WObj:=w7000714;
MoveJ [[330.02,672.74,322.82],[0.584808,0.222494,-0.283349,0.726781],[1,-1,-3,0],[553.979,89.9942,-90.0251,9E+09,9E+09,9E+09]], v600, fine, tPKI500\WObj:=w7000714;

! Keevitus 3.11, h?dromootori plaat, neljas ?mblus, 230 mm, paremalt
MoveJ [[115.44,644.97,326.25],[0.584822,0.222494,-0.283354,0.726768],[1,-1,-3,0],[553.979,89.9942,-90.0251,9E+09,9E+09,9E+09]], v600, fine, tPKI500\WObj:=w7000714;
MoveJ [[118.38,644.59,474.62],[0.63442,0.621795,0.127635,0.441128],[1,-1,-4,0],[553.979,89.9942,-90.0251,9E+09,9E+09,9E+09]], v600, fine, tPKI500\WObj:=w7000714;
ArcLStart [[138.02,630.84,472.29],[0.647181,0.54815,0.031743,0.52885],[1,-1,-4,0],[553.981,89.9942,-90.0254,9E+09,9E+09,9E+09]], v600, seam1, m178job69, fine, tPKI500\WObj:=w7000714;
ArcC [[140.79,629.51,464.42],[0.645735,0.504971,-0.0111766,0.572631],[1,-1,-4,0],[553.98,89.9941,-90.0254,9E+09,9E+09,9E+09]], [[144.16,629.76,456.77],[0.645082,0.458237,-0.0690891,0.607549],[1,-1,-4,0],[553.979,89.9941,-90.0254,9E+09,9E+09,9E+09]], v600, seam1, m178job69, z5, tPKI500\WObj:=w7000714;
ArcL [[170.23,629.83,394.82],[0.626023,0.352436,-0.172535,0.673882],[1,-1,-4,0],[553.982,89.9943,-90.0248,9E+09,9E+09,9E+09]], v600, seam1, m178job69, fine, tPKI500\WObj:=w7000714;
ArcC [[202.39,629.43,359.46],[0.590929,0.239836,-0.267976,0.72213],[1,-1,-3,0],[553.982,89.9942,-90.025,9E+09,9E+09,9E+09]], [[271.56,629.74,330.99],[0.507795,0.0538862,-0.405195,0.758326],[1,-1,-3,0],[553.979,89.9942,-90.0254,9E+09,9E+09,9E+09]], v600, seam1, m178job69, z5, tPKI500\WObj:=w7000714;
ArcCEnd [[301.79,630.62,330.16],[0.381295,-0.145776,-0.534087,0.740348],[1,-1,-3,0],[553.979,89.9942,-90.0248,9E+09,9E+09,9E+09]], [[313.10,628.94,337.94],[0.307156,-0.252191,-0.570662,0.71861],[1,0,-3,0],[553.977,89.9942,-90.0245,9E+09,9E+09,9E+09]], v600, seam1, m178job69, fine, tPKI500\WObj:=w7000714;
MoveJ [[309.94,667.27,318.21],[0.492299,0.0251025,-0.423829,0.759857],[1,-1,-3,0],[553.979,89.9941,-90.0249,9E+09,9E+09,9E+09]], v600, fine, tPKI500\WObj:=w7000714;
MoveJ [[397.45,991.93,334.45],[0.61889,-0.0501983,-0.420622,0.661463],[1,-1,-3,0],[553.978,89.9941,-90.025,9E+09,9E+09,9E+09]], v600, fine, tPKI500\WObj:=w7000714;
GOTO kyljeta2;

! laua p??ramine -60 ja -115 kraadi
MoveJ [[162.45,903.27,491.40],[0.46559,0.241414,-0.541502,0.657056],[0,-1,-3,0],[553.977,59.9851,-115,9E+09,9E+09,9E+09]], v200, fine, tPKI500\WObj:=w7000714;

! Keevitus 3.12, tagant paagi ?mblus, eespool, weavega, 160 mm, paremalt, OK, nurk muutub keevituse alguses
MoveJ [[-43.20,871.48,532.05],[0.359038,0.799285,0.476087,0.0746822],[0,0,-1,0],[553.978,59.9851,-115,9E+09,9E+09,9E+09]], v600, fine, tPKI500\WObj:=w7000714;
MoveJ [[-135.20,821.13,727.31],[0.611943,0.692316,0.348132,0.158209],[0,0,-1,0],[553.979,49.9627,-115,9E+09,9E+09,9E+09]], v600, fine, tPKI500\WObj:=w7000714;
ArcLStart [[-96.63,793.99,748.58],[0.806033,0.530511,0.256844,0.0538631],[0,1,-1,0],[553.982,49.9692,-115,9E+09,9E+09,9E+09]], v600, seam1, wld50v3sh8\Weave:=weave4, fine, tPKI500\WObj:=w7000714;
ArcLEnd [[-151.68,724.68,614.33],[0.86572,0.461946,0.192559,-0.00758197],[0,1,-1,0],[553.979,49.9892,-115,9E+09,9E+09,9E+09]], v600, seam1, wld50v3sh8\Weave:=weave4, fine, tPKI500\WObj:=w7000714;
MoveJ [[-179.72,799.09,528.35],[0.840975,0.494182,0.220255,0.00587413],[0,1,-1,0],[553.978,51.6078,-114.997,9E+09,9E+09,9E+09]], v600, fine, tPKI500\WObj:=w7000714;
MoveJ [[-187.28,803.67,658.32],[0.684096,0.670614,0.286851,0.00272983],[0,0,-1,0],[553.978,59.9853,-115,9E+09,9E+09,9E+09]], v600, fine, tPKI500\WObj:=w7000714;
MoveJ [[-12.20,994.02,708.32],[0.684094,0.670616,0.286851,0.0027351],[0,0,-1,0],[553.978,59.9853,-115,9E+09,9E+09,9E+09]], v600, fine, tPKI500\WObj:=w7000714;

! laua p??ramine -60 ja -70 kraadi
MoveJ [[541.36,1092.26,708.31],[0.633033,0.729356,0.00833812,-0.259307],[0,0,-1,0],[553.977,59.9854,-69.9929,9E+09,9E+09,9E+09]], v200, fine, tPKI500\WObj:=w7000714;

! Keevitus 3.13, eest k?lje ?mblus, tagantpoolt, weavega, 160 mm, paremalt
MoveJ [[750.01,848.15,314.17],[0.633031,0.729357,0.00835907,-0.259312],[0,0,-1,0],[553.977,59.9855,-69.9929,9E+09,9E+09,9E+09]], v600, fine, tPKI500\WObj:=w7000714;
MoveJ [[745.14,802.25,303.86],[0.636213,0.740471,0.0220938,-0.215518],[0,0,-1,0],[553.978,59.9855,-69.9932,9E+09,9E+09,9E+09]], v600, fine, tPKI500\WObj:=w7000714;
ArcLStart [[741.34,784.39,309.70],[0.794022,0.533217,0.0241189,-0.290909],[0,1,-1,0],[553.98,59.9856,-69.9932,9E+09,9E+09,9E+09]], v600, seam1, wld50v3sh8\Weave:=weave4, fine, tPKI500\WObj:=w7000714;
ArcLEnd [[682.53,720.39,184.77],[0.750609,0.631275,0.0326955,-0.192384],[0,1,-1,0],[553.979,59.9854,-69.9931,9E+09,9E+09,9E+09]], v600, seam1, wld50v3sh8\Weave:=weave4, fine, tPKI500\WObj:=w7000714;
MoveJ [[705.58,800.34,225.50],[0.750619,0.631282,0.0325723,-0.192341],[0,0,-1,0],[553.978,59.9856,-69.9933,9E+09,9E+09,9E+09]], v600, fine, tPKI500\WObj:=w7000714;
MoveJ [[866.60,985.78,358.46],[0.750622,0.631276,0.0325848,-0.192344],[0,0,-1,0],[553.977,59.9856,-69.9932,9E+09,9E+09,9E+09]], v600, fine, tPKI500\WObj:=w7000714;
! keevituse nurka muuta 10 kraadi, muidu enam-v?hem [ilus jutt ju!]
kyljeta2:

! laua p??ramine 0 ja 0
MoveJ [[1425.43,552.97,555.84],[0.527174,0.657889,-0.431961,-0.320438],[0,0,-1,0],[553.978,34.2791,-35.2841,9E+09,9E+09,9E+09]], v200, z5, tPKI500\WObj:=w7000714;
MoveJ [[882.55,-78.83,1004.55],[0.208259,0.609785,-0.704636,-0.297119],[0,0,-1,0],[553.978,0.015916,0.016708,9E+09,9E+09,9E+09]], v200, z5, tPKI500\WObj:=w7000714;

! aeg manualis 10:20, 100 % juures
MoveJ [[1148.06,-489.58,1004.56],[0.1324,0.426846,-0.82812,-0.338364],[-1,0,-1,0],[553.977,0.0158778,0.0168768,9E+09,9E+09,9E+09]], v600, z5, tPKI500\WObj:=w7000714;


MoveJ mooduli_vahetus, v600, z50, tPKI500\WObj:=w7000714;

ENDPROC


! tagaots ja paak seest
PROC Tag_paak()

    !Stop;
MoveJ mooduli_vahetus, v600, z50, tPKI500\WObj:=w7000714;

! laua p??ramine 80 ja -20 kraadi
MoveJ [[1813.14,-341.02,-340.35],[0.518989,0.141052,-0.837104,0.10006],[0,-1,0,0],[358.609,79.9979,-19.9396,9E+09,9E+09,9E+09]], v300, z50, tPKI500\WObj:=w7000714;

! Keevitus 4.1, tagant paagi ?mblus, v?limine, 260 mm, paremalt, OK
MoveJ [[1277.77,406.78,343.82],[0.634446,0.593377,-0.468204,-0.161768],[0,-1,0,0],[358.611,79.9979,-19.9396,9E+09,9E+09,9E+09]], v600, z50, tPKI500\WObj:=w7000714;
MoveJ [[1106.16,664.75,466.95],[0.634459,0.59338,-0.468185,-0.16176],[0,-1,0,0],[358.613,79.9981,-19.9396,9E+09,9E+09,9E+09]], v600, z50, tPKI500\WObj:=w7000714;
MoveJ [[1055.61,629.40,456.22],[0.708899,0.588997,-0.370232,-0.116075],[0,-1,0,0],[358.613,79.9981,-19.9396,9E+09,9E+09,9E+09]], v600, z50, tPKI500\WObj:=w7000714;
ArcLStart [[1035.45,620.56,437.43],[0.824577,0.47541,-0.275722,-0.134307],[0,0,0,0],[358.631,79.9998,-19.9384,9E+09,9E+09,9E+09]], v600, seam1, m178job70, fine, tPKI500\WObj:=w7000714;
ArcL [[1009.87,622.25,387.87],[0.787027,0.55501,-0.250654,-0.0986254],[0,0,0,0],[358.615,79.9985,-19.9399,9E+09,9E+09,9E+09]], v600, seam1, m178job70, fine, tPKI500\WObj:=w7000714;
ArcL [[995.71,624.48,359.17],[0.797513,0.574666,-0.160933,-0.0885156],[0,0,0,0],[358.604,79.9983,-19.9404,9E+09,9E+09,9E+09]], v600, seam1, m178job70, fine, tPKI500\WObj:=w7000714;
ArcL [[985.56,624.28,340.01],[0.773128,0.598545,-0.124705,-0.168721],[0,0,-1,0],[460.305,73.7027,-18.3705,9E+09,9E+09,9E+09]], v600, seam1, m178job70, fine, tPKI500\WObj:=w7000714;
ArcL [[950.79,627.22,272.25],[0.841528,0.527105,-0.0802795,-0.08688],[0,0,0,0],[358.587,79.9986,-19.9548,9E+09,9E+09,9E+09]], v600, seam1, m178job70, fine, tPKI500\WObj:=w7000714;
ArcL [[939.60,626.97,249.02],[0.838126,0.518781,-0.123641,-0.114565],[0,0,0,0],[358.596,79.9988,-19.9542,9E+09,9E+09,9E+09]], v600, seam1, m178job70, fine, tPKI500\WObj:=w7000714;
ArcL [[931.60,627.03,234.71],[0.849343,0.489535,-0.0896768,-0.175875],[0,0,-1,0],[358.589,79.9987,-19.9547,9E+09,9E+09,9E+09]], v600, seam1, m178job70, fine, tPKI500\WObj:=w7000714;
!ArcL [[922.20,625.23,220.08],[0.849298,0.489491,-0.0899854,-0.176058],[0,0,-1,0],[358.594,79.9989,-19.9551,9E+09,9E+09,9E+09]], v600, seam1, wld100v4sh16, z5, tPKI500\WObj:=w7000714;
ArcLEnd [[920.38,624.98,214.95],[0.849325,0.489559,-0.0896895,-0.175887],[0,0,-1,0],[358.606,79.999,-19.954,9E+09,9E+09,9E+09]], v600, seam1, m178job70, fine, tPKI500\WObj:=w7000714;
MoveJ [[946.78,697.13,173.80],[0.716876,0.60114,-0.339611,-0.0968779],[0,-1,0,0],[358.613,79.9982,-19.9402,9E+09,9E+09,9E+09]], v600, z5, tPKI500\WObj:=w7000714;
!Stop;
MoveJ [[1045.27,688.20,245.16],[0.716875,0.601131,-0.339627,-0.0968855],[0,-1,0,0],[358.61,79.9981,-19.9402,9E+09,9E+09,9E+09]], v600, z5, tPKI500\WObj:=w7000714;

! Keevitus 4.2, tagant paagi ?mblus, sisemine, 95+120+20 mm, vasakult, OK
MoveJ [[1170.61,334.72,242.62],[0.688602,0.568129,-0.405118,-0.197327],[0,0,-1,0],[358.611,79.9982,-19.9402,9E+09,9E+09,9E+09]], v600, z5, tPKI500\WObj:=w7000714;
MoveJ [[1006.85,163.11,357.36],[0.79716,0.508494,-0.268825,-0.183588],[0,0,-1,0],[358.61,79.9983,-19.9402,9E+09,9E+09,9E+09]], v600, z5, tPKI500\WObj:=w7000714;
ArcLStart [[971.01,126.32,395.63],[0.796905,0.508931,-0.268677,-0.1837],[0,0,0,0],[358.619,79.9987,-19.9404,9E+09,9E+09,9E+09]], v600, seam1, m178job70, fine, tPKI500\WObj:=w7000714;
ArcL [[935.89,127.49,323.60],[0.79466,0.512431,-0.271175,-0.179987],[0,0,-1,0],[358.62,79.9984,-19.9396,9E+09,9E+09,9E+09]], v600, seam1, m178job70, fine, tPKI500\WObj:=w7000714;
!ArcL [[933.20,127.56,326.62],[0.794936,0.512007,-0.271255,-0.179855],[0,0,-1,0],[358.612,79.9987,-19.9399,9E+09,9E+09,9E+09]], v600, seam1, wld100v4sh16, fine, tPKI500\WObj:=w7000714;
ArcL [[929.13,128.99,252.15],[0.792223,0.513572,-0.20681,-0.256627],[0,0,-1,0],[358.614,79.9987,-19.9409,9E+09,9E+09,9E+09]], v600, seam1, m178job70, fine, tPKI500\WObj:=w7000714;
ArcL [[926.36,128.21,221.48],[0.878581,0.360035,-0.281748,-0.138167],[0,0,0,0],[358.579,79.999,-19.9422,9E+09,9E+09,9E+09]], v600, seam1, m178job70, fine, tPKI500\WObj:=w7000714;
ArcL [[923.62,128.14,218.22],[0.878583,0.360044,-0.281727,-0.138172],[0,0,0,0],[358.594,79.9993,-19.9416,9E+09,9E+09,9E+09]], v600, seam1, m178job70, fine, tPKI500\WObj:=w7000714;
ArcLEnd [[920.25,128.85,213.47],[0.878526,0.360168,-0.281738,-0.13819],[0,0,0,0],[358.594,79.999,-19.9414,9E+09,9E+09,9E+09]], v600, seam1, m178job70, fine, tPKI500\WObj:=w7000714;
MoveJ [[916.53,135.19,190.85],[0.932968,0.216189,-0.267507,-0.106178],[0,0,0,0],[358.612,79.9985,-19.9404,9E+09,9E+09,9E+09]], v600, z5, tPKI500\WObj:=w7000714;
!Stop;
MoveJ [[1075.67,191.40,221.02],[0.932964,0.216201,-0.267512,-0.106181],[0,0,0,0],[358.612,79.9985,-19.9402,9E+09,9E+09,9E+09]], v600, z5, tPKI500\WObj:=w7000714;

! laua p??ramine 80 ja 20 kraadi
MoveJ [[863.32,-235.23,233.81],[0.840658,0.111885,-0.325241,-0.418325],[0,0,0,0],[358.612,79.9987,19.9855,9E+09,9E+09,9E+09]], v200, z5, tPKI500\WObj:=w7000714;

! Keevitus 4.3, tagant paagi ?mblus, sisemine, 95+120+20 mm, paremalt, OK
MoveJ [[1123.65,95.51,356.45],[0.840753,0.111905,-0.32513,-0.418215],[0,0,0,0],[358.613,79.9987,19.9855,9E+09,9E+09,9E+09]], v600, z5, tPKI500\WObj:=w7000714;
MoveJ [[1110.51,428.94,284.26],[0.805836,-0.382676,-0.320423,-0.31862],[0,-1,1,0],[358.612,79.9987,19.9856,9E+09,9E+09,9E+09]], v600, z5, tPKI500\WObj:=w7000714;
MoveJ [[1006.23,571.97,381.60],[0.803339,-0.367161,-0.382698,-0.270891],[0,-1,1,0],[358.613,79.9987,19.9855,9E+09,9E+09,9E+09]], v600, z5, tPKI500\WObj:=w7000714;
ArcLStart [[974.01,603.01,399.65],[0.826326,-0.271663,-0.408595,-0.27647],[0,-1,1,0],[358.633,79.9998,19.9828,9E+09,9E+09,9E+09]], v600, seam1, m178job70, fine, tPKI500\WObj:=w7000714;
ArcL [[937.98,603.78,327.86],[0.792053,-0.272924,-0.467261,-0.282548],[0,-1,1,0],[358.622,79.9996,19.9841,9E+09,9E+09,9E+09]], v600, seam1, m178job70, fine, tPKI500\WObj:=w7000714;
ArcL [[930.89,604.98,254.48],[0.762195,-0.273647,-0.510164,-0.289673],[0,-1,1,0],[358.604,79.9998,19.9843,9E+09,9E+09,9E+09]], v600, seam1, m178job70, fine, tPKI500\WObj:=w7000714;
ArcL [[928.18,605.49,227.69],[0.788549,-0.273139,-0.472401,-0.28359],[0,-1,1,0],[358.649,79.9997,19.9855,9E+09,9E+09,9E+09]], v600, seam1, m178job70, fine, tPKI500\WObj:=w7000714;
!ArcL [[921.65,607.63,218.71],[0.909227,-0.123785,-0.301158,-0.259401],[0,-1,0,0],[358.611,79.9987,19.9858,9E+09,9E+09,9E+09]], v600, seam1, wld100v4sh16, fine, tPKI500\WObj:=w7000714;
ArcLEnd [[920.83,606.71,220.46],[0.788588,-0.273122,-0.472387,-0.283523],[0,-1,1,0],[358.65,80,19.9846,9E+09,9E+09,9E+09]], v600, seam1, m178job70, fine, tPKI500\WObj:=w7000714;
MoveJ [[927.14,599.07,202.42],[0.894134,-0.126995,-0.341679,-0.260102],[0,-1,0,0],[358.613,79.9987,19.9856,9E+09,9E+09,9E+09]], v600, z5, tPKI500\WObj:=w7000714;
!Stop;
MoveJ [[1082.56,312.66,248.06],[0.894138,-0.126993,-0.341676,-0.260093],[0,-1,0,0],[358.611,79.9987,19.9856,9E+09,9E+09,9E+09]], v600, z5, tPKI500\WObj:=w7000714;

! Keevitus 4.4, tagant paagi ?mblus, v?limine, 260 mm, vasakult, OK
MoveJ [[1102.60,-17.06,440.83],[0.894757,-0.111448,-0.343068,-0.26324],[0,-1,0,0],[358.612,79.9987,19.9857,9E+09,9E+09,9E+09]], v600, z5, tPKI500\WObj:=w7000714;
MoveJ [[1030.08,10.02,426.99],[0.833295,-0.432352,-0.298391,-0.172206],[0,-1,1,0],[358.612,79.9988,19.9855,9E+09,9E+09,9E+09]], v600, z5, tPKI500\WObj:=w7000714;
ArcLStart [[1027.59,107.27,438.64],[0.833468,-0.432257,-0.298407,-0.171582],[0,-1,1,0],[358.618,79.9994,19.9867,9E+09,9E+09,9E+09]], v600, seam1, m178job70, fine, tPKI500\WObj:=w7000714;
ArcL [[1001.63,106.87,386.31],[0.833437,-0.432271,-0.298387,-0.171729],[0,-1,1,0],[358.622,79.9993,19.9834,9E+09,9E+09,9E+09]], v600, seam1, m178job70, fine, tPKI500\WObj:=w7000714;
ArcL [[991.27,105.66,364.38],[0.814371,-0.451347,-0.289393,-0.222122],[0,-1,1,0],[358.619,79.9987,19.9857,9E+09,9E+09,9E+09]], v600, seam1, m178job70, fine, tPKI500\WObj:=w7000714;
ArcL [[932.80,107.34,250.67],[0.811101,-0.470959,-0.275966,-0.210137],[0,-1,1,0],[358.618,79.9987,19.986,9E+09,9E+09,9E+09]], v600, seam1, m178job70, fine, tPKI500\WObj:=w7000714;
ArcLEnd [[915.94,107.06,215.57],[0.821101,-0.442565,-0.315082,-0.175082],[0,-1,1,0],[358.618,79.9987,19.9851,9E+09,9E+09,9E+09]], v600, seam1, m178job70, fine, tPKI500\WObj:=w7000714;
MoveJ [[930.78,81.45,225.70],[0.820989,-0.442623,-0.315085,-0.175456],[0,-1,1,0],[358.613,79.9988,19.9854,9E+09,9E+09,9E+09]], v600, z5, tPKI500\WObj:=w7000714;
!Stop;
MoveJ [[1155.64,-71.28,272.47],[0.820996,-0.442609,-0.315089,-0.175452],[0,-1,1,0],[358.611,79.9988,19.9854,9E+09,9E+09,9E+09]], v600, z5, tPKI500\WObj:=w7000714;

! laua p??ramine 0 ja 0 kraadi
MoveJ [[311.03,89.38,1075.54],[0.391937,-0.277108,-0.835687,-0.266879],[0,-1,1,0],[358.614,-0.000860473,-0.00206977,9E+09,9E+09,9E+09]], v200, z5, tPKI500\WObj:=w7000714;
!Stop;

